gfCNCPoint2[23989] = {X 180.1466, Y 22.4199, Z -3.0000, A 0.000, B 0.000, C 0.000 }
gfCNCPoint2[23990] = {X 179.6136, Y 22.9696, Z -3.0000, A 0.000, B 0.000, C 0.000 }
gfCNCPoint2[23991] = {X 180.2003, Y 22.9879, Z -3.0000, A 0.000, B 0.000, C 0.000 }
gfCNCPoint2[23992] = {X 182.2741, Y 22.7679, Z -3.0000, A 0.000, B 0.000, C 0.000 }
gfCNCPoint2[23993] = {X 184.3552, Y 22.6339, Z -3.0000, A 0.000, B 0.000, C 0.000 }
gfCNCPoint2[23994] = {X 184.7920, Y 22.6180, Z -3.0000, A 0.000, B 0.000, C 0.000 }
gfCNCPoint2[23995] = {X 185.2288, Y 22.6003, Z -3.0000, A 0.000, B 0.000, C 0.000 }
gfCNCPoint2[23996] = {X 185.1444, Y 20.6021, Z -3.0000, A 0.000, B 0.000, C 0.000 }
gfCNCPoint2[23997] = {X 185.1444, Y 20.6021, Z 0.0000, A 0.000, B 0.000, C 0.000 }
gfCNCPoint2[23998] = {X 185.1444, Y 20.6021, Z 11.0000, A 0.000, B 0.000, C 0.000 }
gfCNCPoint2[23999] = {X 186.2306, Y 37.9128, Z 11.0000, A 0.000, B 0.000, C 0.000 }
gfCNCPoint2[24000] = {X 186.2306, Y 37.9128, Z 0.8333, A 0.000, B 0.000, C 0.000 }
gfCNCPoint2[24001] = {X 187.5931, Y 37.8326, Z 0.4676, A 0.000, B 0.000, C 0.000 }
gfCNCPoint2[24002] = {X 189.4216, Y 37.3852, Z -0.0368, A 0.000, B 0.000, C 0.000 }
gfCNCPoint2[24003] = {X 190.1467, Y 37.0730, Z -0.2483, A 0.000, B 0.000, C 0.000 }
gfCNCPoint2[24004] = {X 190.9837, Y 36.7127, Z -0.4925, A 0.000, B 0.000, C 0.000 }
gfCNCPoint2[24005] = {X 191.6928, Y 36.3239, Z -0.7092, A 0.000, B 0.000, C 0.000 }
gfCNCPoint2[24006] = {X 192.4466, Y 35.8119, Z -0.9533, A 0.000, B 0.000, C 0.000 }
gfCNCPoint2[24007] = {X 192.4699, Y 35.2978, Z -1.0913, A 0.000, B 0.000, C 0.000 }
gfCNCPoint2[24008] = {X 192.6316, Y 34.6339, Z -1.2743, A 0.000, B 0.000, C 0.000 }
gfCNCPoint2[24009] = {X 192.8474, Y 34.1666, Z -1.4123, A 0.000, B 0.000, C 0.000 }
gfCNCPoint2[24010] = {X 192.7390, Y 34.1918, Z -1.4421, A 0.000, B 0.000, C 0.000 }
gfCNCPoint2[24011] = {X 191.4103, Y 34.4420, Z -1.8044, A 0.000, B 0.000, C 0.000 }
gfCNCPoint2[24012] = {X 190.5793, Y 34.5489, Z -2.0289, A 0.000, B 0.000, C 0.000 }
gfCNCPoint2[24013] = {X 189.2271, Y 34.6435, Z -2.3921, A 0.000, B 0.000, C 0.000 }
gfCNCPoint2[24014] = {X 186.9625, Y 34.7826, Z -3.0000, A 0.000, B 0.000, C 0.000 }
gfCNCPoint2[24015] = {X 182.5767, Y 35.0519, Z -3.0000, A 0.000, B 0.000, C 0.000 }
gfCNCPoint2[24016] = {X 181.8176, Y 35.1394, Z -3.0000, A 0.000, B 0.000, C 0.000 }
gfCNCPoint2[24017] = {X 181.0723, Y 35.3075, Z -3.0000, A 0.000, B 0.000, C 0.000 }
gfCNCPoint2[24018] = {X 181.0641, Y 35.3819, Z -3.0000, A 0.000, B 0.000, C 0.000 }
gfCNCPoint2[24019] = {X 181.0641, Y 35.4568, Z -3.0000, A 0.000, B 0.000, C 0.000 }
gfCNCPoint2[24020] = {X 181.1571, Y 36.0001, Z -3.0000, A 0.000, B 0.000, C 0.000 }
gfCNCPoint2[24021] = {X 181.4145, Y 36.4875, Z -3.0000, A 0.000, B 0.000, C 0.000 }
gfCNCPoint2[24022] = {X 181.8107, Y 36.8707, Z -3.0000, A 0.000, B 0.000, C 0.000 }
gfCNCPoint2[24023] = {X 182.4285, Y 37.2234, Z -3.0000, A 0.000, B 0.000, C 0.000 }
gfCNCPoint2[24024] = {X 183.0887, Y 37.4882, Z -3.0000, A 0.000, B 0.000, C 0.000 }
gfCNCPoint2[24025] = {X 184.4959, Y 37.8021, Z -3.0000, A 0.000, B 0.000, C 0.000 }
gfCNCPoint2[24026] = {X 185.9331, Y 37.9178, Z -3.0000, A 0.000, B 0.000, C 0.000 }
gfCNCPoint2[24027] = {X 187.3724, Y 37.8332, Z -3.0000, A 0.000, B 0.000, C 0.000 }
gfCNCPoint2[24028] = {X 188.7860, Y 37.5497, Z -3.0000, A 0.000, B 0.000, C 0.000 }
gfCNCPoint2[24029] = {X 190.1467, Y 37.0730, Z -3.0000, A 0.000, B 0.000, C 0.000 }
gfCNCPoint2[24030] = {X 191.3267, Y 36.4971, Z -3.0000, A 0.000, B 0.000, C 0.000 }
gfCNCPoint2[24031] = {X 192.4466, Y 35.8119, Z -3.0000, A 0.000, B 0.000, C 0.000 }
gfCNCPoint2[24032] = {X 192.5671, Y 34.9698, Z -3.0000, A 0.000, B 0.000, C 0.000 }
gfCNCPoint2[24033] = {X 192.8474, Y 34.1666, Z -3.0000, A 0.000, B 0.000, C 0.000 }
gfCNCPoint2[24034] = {X 192.7390, Y 34.1918, Z -3.0000, A 0.000, B 0.000, C 0.000 }
gfCNCPoint2[24035] = {X 190.9896, Y 34.4688, Z -3.0000, A 0.000, B 0.000, C 0.000 }
gfCNCPoint2[24036] = {X 189.2271, Y 34.6435, Z -3.0000, A 0.000, B 0.000, C 0.000 }
gfCNCPoint2[24037] = {X 186.9625, Y 34.7826, Z -3.0000, A 0.000, B 0.000, C 0.000 }
gfCNCPoint2[24038] = {X 190.9563, Y 34.8065, Z -3.0000, A 0.000, B 0.000, C 0.000 }
gfCNCPoint2[24039] = {X 186.9576, Y 34.7027, Z -3.0000, A 0.000, B 0.000, C 0.000 }
gfCNCPoint2[24040] = {X 182.5718, Y 34.9720, Z -3.0000, A 0.000, B 0.000, C 0.000 }
gfCNCPoint2[24041] = {X 181.7801, Y 35.0647, Z -3.0000, A 0.000, B 0.000, C 0.000 }
gfCNCPoint2[24042] = {X 181.0034, Y 35.2440, Z -3.0000, A 0.000, B 0.000, C 0.000 }
gfCNCPoint2[24043] = {X 180.9865, Y 35.3479, Z -3.0000, A 0.000, B 0.000, C 0.000 }
gfCNCPoint2[24044] = {X 180.9840, Y 35.4530, Z -3.0000, A 0.000, B 0.000, C 0.000 }
gfCNCPoint2[24045] = {X 181.0805, Y 36.0232, Z -3.0000, A 0.000, B 0.000, C 0.000 }
gfCNCPoint2[24046] = {X 181.3499, Y 36.5348, Z -3.0000, A 0.000, B 0.000, C 0.000 }
gfCNCPoint2[24047] = {X 181.7656, Y 36.9368, Z -3.0000, A 0.000, B 0.000, C 0.000 }
gfCNCPoint2[24048] = {X 182.3937, Y 37.2955, Z -3.0000, A 0.000, B 0.000, C 0.000 }
gfCNCPoint2[24049] = {X 183.0650, Y 37.5647, Z -3.0000, A 0.000, B 0.000, C 0.000 }
gfCNCPoint2[24050] = {X 184.4832, Y 37.8811, Z -3.0000, A 0.000, B 0.000, C 0.000 }
gfCNCPoint2[24051] = {X 185.9316, Y 37.9978, Z -3.0000, A 0.000, B 0.000, C 0.000 }
gfCNCPoint2[24052] = {X 187.3822, Y 37.9125, Z -3.0000, A 0.000, B 0.000, C 0.000 }
gfCNCPoint2[24053] = {X 188.8070, Y 37.6269, Z -3.0000, A 0.000, B 0.000, C 0.000 }
gfCNCPoint2[24054] = {X 190.1784, Y 37.1465, Z -3.0000, A 0.000, B 0.000, C 0.000 }
gfCNCPoint2[24055] = {X 191.3828, Y 36.5576, Z -3.0000, A 0.000, B 0.000, C 0.000 }
gfCNCPoint2[24056] = {X 192.5249, Y 35.8554, Z -3.0000, A 0.000, B 0.000, C 0.000 }
gfCNCPoint2[24057] = {X 192.6603, Y 34.9271, Z -3.0000, A 0.000, B 0.000, C 0.000 }
gfCNCPoint2[24058] = {X 192.9929, Y 34.0499, Z -3.0000, A 0.000, B 0.000, C 0.000 }
gfCNCPoint2[24059] = {X 192.7315, Y 34.1118, Z -3.0000, A 0.000, B 0.000, C 0.000 }
gfCNCPoint2[24060] = {X 190.9841, Y 34.3888, Z -3.0000, A 0.000, B 0.000, C 0.000 }
gfCNCPoint2[24061] = {X 189.2235, Y 34.5636, Z -3.0000, A 0.000, B 0.000, C 0.000 }
gfCNCPoint2[24062] = {X 186.9576, Y 34.7027, Z -3.0000, A 0.000, B 0.000, C 0.000 }
gfCNCPoint2[24063] = {X 183.0017, Y 35.2949, Z -3.0000, A 0.000, B 0.000, C 0.000 }
gfCNCPoint2[24064] = {X 190.9514, Y 34.7266, Z -3.0000, A 0.000, B 0.000, C 0.000 }
gfCNCPoint2[24065] = {X 186.9527, Y 34.6229, Z -3.0000, A 0.000, B 0.000, C 0.000 }
gfCNCPoint2[24066] = {X 182.5669, Y 34.8922, Z -3.0000, A 0.000, B 0.000, C 0.000 }
gfCNCPoint2[24067] = {X 181.7440, Y 34.9898, Z -3.0000, A 0.000, B 0.000, C 0.000 }
gfCNCPoint2[24068] = {X 180.9376, Y 35.1800, Z -3.0000, A 0.000, B 0.000, C 0.000 }
gfCNCPoint2[24069] = {X 180.9095, Y 35.3162, Z -3.0000, A 0.000, B 0.000, C 0.000 }
gfCNCPoint2[24070] = {X 180.9041, Y 35.4551, Z -3.0000, A 0.000, B 0.000, C 0.000 }
gfCNCPoint2[24071] = {X 181.0051, Y 36.0500, Z -3.0000, A 0.000, B 0.000, C 0.000 }
gfCNCPoint2[24072] = {X 181.2866, Y 36.5836, Z -3.0000, A 0.000, B 0.000, C 0.000 }
gfCNCPoint2[24073] = {X 181.7205, Y 37.0029, Z -3.0000, A 0.000, B 0.000, C 0.000 }
gfCNCPoint2[24074] = {X 182.3589, Y 37.3675, Z -3.0000, A 0.000, B 0.000, C 0.000 }
gfCNCPoint2[24075] = {X 183.0413, Y 37.6411, Z -3.0000, A 0.000, B 0.000, C 0.000 }
gfCNCPoint2[24076] = {X 184.4705, Y 37.9601, Z -3.0000, A 0.000, B 0.000, C 0.000 }
gfCNCPoint2[24077] = {X 185.9302, Y 38.0778, Z -3.0000, A 0.000, B 0.000, C 0.000 }
gfCNCPoint2[24078] = {X 187.3921, Y 37.9919, Z -3.0000, A 0.000, B 0.000, C 0.000 }
gfCNCPoint2[24079] = {X 188.8279, Y 37.7041, Z -3.0000, A 0.000, B 0.000, C 0.000 }
gfCNCPoint2[24080] = {X 190.2100, Y 37.2200, Z -3.0000, A 0.000, B 0.000, C 0.000 }
gfCNCPoint2[24081] = {X 191.4392, Y 36.6179, Z -3.0000, A 0.000, B 0.000, C 0.000 }
gfCNCPoint2[24082] = {X 192.6036, Y 35.8985, Z -3.0000, A 0.000, B 0.000, C 0.000 }
gfCNCPoint2[24083] = {X 192.6773, Y 35.2160, Z -3.0000, A 0.000, B 0.000, C 0.000 }
gfCNCPoint2[24084] = {X 192.8602, Y 34.5544, Z -3.0000, A 0.000, B 0.000, C 0.000 }
gfCNCPoint2[24085] = {X 193.1474, Y 33.9310, Z -3.0000, A 0.000, B 0.000, C 0.000 }
gfCNCPoint2[24086] = {X 192.7149, Y 34.0336, Z -3.0000, A 0.000, B 0.000, C 0.000 }
gfCNCPoint2[24087] = {X 190.9732, Y 34.3096, Z -3.0000, A 0.000, B 0.000, C 0.000 }
gfCNCPoint2[24088] = {X 189.2183, Y 34.4838, Z -3.0000, A 0.000, B 0.000, C 0.000 }
gfCNCPoint2[24089] = {X 186.9527, Y 34.6229, Z -3.0000, A 0.000, B 0.000, C 0.000 }
gfCNCPoint2[24090] = {X 182.9968, Y 35.2151, Z -3.0000, A 0.000, B 0.000, C 0.000 }
gfCNCPoint2[24091] = {X 190.9465, Y 34.6468, Z -3.0000, A 0.000, B 0.000, C 0.000 }
gfCNCPoint2[24092] = {X 186.9478, Y 34.5430, Z -3.0000, A 0.000, B 0.000, C 0.000 }
gfCNCPoint2[24093] = {X 182.5620, Y 34.8123, Z -3.0000, A 0.000, B 0.000, C 0.000 }
gfCNCPoint2[24094] = {X 181.7093, Y 34.9147, Z -3.0000, A 0.000, B 0.000, C 0.000 }
gfCNCPoint2[24095] = {X 180.8742, Y 35.1154, Z -3.0000, A 0.000, B 0.000, C 0.000 }
gfCNCPoint2[24096] = {X 180.8331, Y 35.2840, Z -3.0000, A 0.000, B 0.000, C 0.000 }
gfCNCPoint2[24097] = {X 180.8241, Y 35.4572, Z -3.0000, A 0.000, B 0.000, C 0.000 }
gfCNCPoint2[24098] = {X 180.9297, Y 36.0768, Z -3.0000, A 0.000, B 0.000, C 0.000 }
gfCNCPoint2[24099] = {X 181.2232, Y 36.6325, Z -3.0000, A 0.000, B 0.000, C 0.000 }
gfCNCPoint2[24100] = {X 181.6754, Y 37.0690, Z -3.0000, A 0.000, B 0.000, C 0.000 }
gfCNCPoint2[24101] = {X 182.3241, Y 37.4395, Z -3.0000, A 0.000, B 0.000, C 0.000 }
gfCNCPoint2[24102] = {X 183.0176, Y 37.7175, Z -3.0000, A 0.000, B 0.000, C 0.000 }
gfCNCPoint2[24103] = {X 184.4578, Y 38.0391, Z -3.0000, A 0.000, B 0.000, C 0.000 }
gfCNCPoint2[24104] = {X 185.9288, Y 38.1578, Z -3.0000, A 0.000, B 0.000, C 0.000 }
gfCNCPoint2[24105] = {X 187.4020, Y 38.0713, Z -3.0000, A 0.000, B 0.000, C 0.000 }
gfCNCPoint2[24106] = {X 188.8489, Y 37.7813, Z -3.0000, A 0.000, B 0.000, C 0.000 }
gfCNCPoint2[24107] = {X 190.2416, Y 37.2935, Z -3.0000, A 0.000, B 0.000, C 0.000 }
gfCNCPoint2[24108] = {X 191.4958, Y 36.6780, Z -3.0000, A 0.000, B 0.000, C 0.000 }
gfCNCPoint2[24109] = {X 192.6827, Y 35.9411, Z -3.0000, A 0.000, B 0.000, C 0.000 }
gfCNCPoint2[24110] = {X 192.7627, Y 35.1965, Z -3.0000, A 0.000, B 0.000, C 0.000 }
gfCNCPoint2[24111] = {X 192.9748, Y 34.4783, Z -3.0000, A 0.000, B 0.000, C 0.000 }
gfCNCPoint2[24112] = {X 193.3123, Y 33.8097, Z -3.0000, A 0.000, B 0.000, C 0.000 }
gfCNCPoint2[24113] = {X 192.6983, Y 33.9553, Z -3.0000, A 0.000, B 0.000, C 0.000 }
gfCNCPoint2[24114] = {X 190.9622, Y 34.2303, Z -3.0000, A 0.000, B 0.000, C 0.000 }
gfCNCPoint2[24115] = {X 189.2131, Y 34.4039, Z -3.0000, A 0.000, B 0.000, C 0.000 }
gfCNCPoint2[24116] = {X 186.9478, Y 34.5430, Z -3.0000, A 0.000, B 0.000, C 0.000 }
gfCNCPoint2[24117] = {X 182.9919, Y 35.1352, Z -3.0000, A 0.000, B 0.000, C 0.000 }
gfCNCPoint2[24118] = {X 190.9415, Y 34.5669, Z -3.0000, A 0.000, B 0.000, C 0.000 }
gfCNCPoint2[24119] = {X 186.9429, Y 34.4632, Z -3.0000, A 0.000, B 0.000, C 0.000 }
gfCNCPoint2[24120] = {X 182.5571, Y 34.7325, Z -3.0000, A 0.000, B 0.000, C 0.000 }
gfCNCPoint2[24121] = {X 181.6755, Y 34.8395, Z -3.0000, A 0.000, B 0.000, C 0.000 }
gfCNCPoint2[24122] = {X 180.8129, Y 35.0505, Z -3.0000, A 0.000, B 0.000, C 0.000 }
gfCNCPoint2[24123] = {X 180.7572, Y 35.2513, Z -3.0000, A 0.000, B 0.000, C 0.000 }
gfCNCPoint2[24124] = {X 180.7441, Y 35.4593, Z -3.0000, A 0.000, B 0.000, C 0.000 }
gfCNCPoint2[24125] = {X 180.8543, Y 36.1035, Z -3.0000, A 0.000, B 0.000, C 0.000 }
gfCNCPoint2[24126] = {X 181.1598, Y 36.6813, Z -3.0000, A 0.000, B 0.000, C 0.000 }
gfCNCPoint2[24127] = {X 181.6303, Y 37.1351, Z -3.0000, A 0.000, B 0.000, C 0.000 }
gfCNCPoint2[24128] = {X 182.2893, Y 37.5116, Z -3.0000, A 0.000, B 0.000, C 0.000 }
gfCNCPoint2[24129] = {X 182.9939, Y 37.7939, Z -3.0000, A 0.000, B 0.000, C 0.000 }
gfCNCPoint2[24130] = {X 184.4452, Y 38.1181, Z -3.0000, A 0.000, B 0.000, C 0.000 }
gfCNCPoint2[24131] = {X 185.9274, Y 38.2378, Z -3.0000, A 0.000, B 0.000, C 0.000 }
gfCNCPoint2[24132] = {X 187.4118, Y 38.1507, Z -3.0000, A 0.000, B 0.000, C 0.000 }
gfCNCPoint2[24133] = {X 188.8699, Y 37.8585, Z -3.0000, A 0.000, B 0.000, C 0.000 }
gfCNCPoint2[24134] = {X 190.2733, Y 37.3669, Z -3.0000, A 0.000, B 0.000, C 0.000 }
gfCNCPoint2[24135] = {X 191.5527, Y 36.7379, Z -3.0000, A 0.000, B 0.000, C 0.000 }
gfCNCPoint2[24136] = {X 192.7622, Y 35.9833, Z -3.0000, A 0.000, B 0.000, C 0.000 }
gfCNCPoint2[24137] = {X 192.8359, Y 35.2389, Z -3.0000, A 0.000, B 0.000, C 0.000 }
gfCNCPoint2[24138] = {X 193.0442, Y 34.5204, Z -3.0000, A 0.000, B 0.000, C 0.000 }
gfCNCPoint2[24139] = {X 193.3801, Y 33.8520, Z -3.0000, A 0.000, B 0.000, C 0.000 }
gfCNCPoint2[24140] = {X 193.4231, Y 33.7847, Z -3.0000, A 0.000, B 0.000, C 0.000 }
gfCNCPoint2[24141] = {X 193.4673, Y 33.7182, Z -3.0000, A 0.000, B 0.000, C 0.000 }
gfCNCPoint2[24142] = {X 193.3655, Y 33.7149, Z -3.0000, A 0.000, B 0.000, C 0.000 }
gfCNCPoint2[24143] = {X 192.6816, Y 33.8770, Z -3.0000, A 0.000, B 0.000, C 0.000 }
gfCNCPoint2[24144] = {X 190.9512, Y 34.1511, Z -3.0000, A 0.000, B 0.000, C 0.000 }
gfCNCPoint2[24145] = {X 189.2078, Y 34.3241, Z -3.0000, A 0.000, B 0.000, C 0.000 }
gfCNCPoint2[24146] = {X 186.9429, Y 34.4632, Z -3.0000, A 0.000, B 0.000, C 0.000 }
gfCNCPoint2[24147] = {X 182.9870, Y 35.0554, Z -3.0000, A 0.000, B 0.000, C 0.000 }
gfCNCPoint2[24148] = {X 190.9366, Y 34.4871, Z -3.0000, A 0.000, B 0.000, C 0.000 }
gfCNCPoint2[24149] = {X 186.9380, Y 34.3833, Z -3.0000, A 0.000, B 0.000, C 0.000 }
gfCNCPoint2[24150] = {X 182.5522, Y 34.6526, Z -3.0000, A 0.000, B 0.000, C 0.000 }
gfCNCPoint2[24151] = {X 181.6426, Y 34.7642, Z -3.0000, A 0.000, B 0.000, C 0.000 }
gfCNCPoint2[24152] = {X 180.7533, Y 34.9853, Z -3.0000, A 0.000, B 0.000, C 0.000 }
gfCNCPoint2[24153] = {X 180.6819, Y 35.2183, Z -3.0000, A 0.000, B 0.000, C 0.000 }
gfCNCPoint2[24154] = {X 180.6641, Y 35.4613, Z -3.0000, A 0.000, B 0.000, C 0.000 }
gfCNCPoint2[24155] = {X 180.7789, Y 36.1303, Z -3.0000, A 0.000, B 0.000, C 0.000 }
gfCNCPoint2[24156] = {X 181.0965, Y 36.7302, Z -3.0000, A 0.000, B 0.000, C 0.000 }
gfCNCPoint2[24157] = {X 181.5852, Y 37.2012, Z -3.0000, A 0.000, B 0.000, C 0.000 }
gfCNCPoint2[24158] = {X 182.2546, Y 37.5836, Z -3.0000, A 0.000, B 0.000, C 0.000 }
gfCNCPoint2[24159] = {X 182.9702, Y 37.8703, Z -3.0000, A 0.000, B 0.000, C 0.000 }
gfCNCPoint2[24160] = {X 184.4325, Y 38.1971, Z -3.0000, A 0.000, B 0.000, C 0.000 }
gfCNCPoint2[24161] = {X 185.9259, Y 38.3178, Z -3.0000, A 0.000, B 0.000, C 0.000 }
gfCNCPoint2[24162] = {X 187.4217, Y 38.2301, Z -3.0000, A 0.000, B 0.000, C 0.000 }
gfCNCPoint2[24163] = {X 188.8908, Y 37.9358, Z -3.0000, A 0.000, B 0.000, C 0.000 }
gfCNCPoint2[24164] = {X 190.3049, Y 37.4404, Z -3.0000, A 0.000, B 0.000, C 0.000 }
gfCNCPoint2[24165] = {X 191.6098, Y 36.7977, Z -3.0000, A 0.000, B 0.000, C 0.000 }
gfCNCPoint2[24166] = {X 192.8422, Y 36.0250, Z -3.0000, A 0.000, B 0.000, C 0.000 }
gfCNCPoint2[24167] = {X 192.9290, Y 35.1818, Z -3.0000, A 0.000, B 0.000, C 0.000 }
gfCNCPoint2[24168] = {X 193.1917, Y 34.3757, Z -3.0000, A 0.000, B 0.000, C 0.000 }
gfCNCPoint2[24169] = {X 193.6183, Y 33.6431, Z -3.0000, A 0.000, B 0.000, C 0.000 }
gfCNCPoint2[24170] = {X 193.3575, Y 33.6346, Z -3.0000, A 0.000, B 0.000, C 0.000 }
gfCNCPoint2[24171] = {X 192.6650, Y 33.7987, Z -3.0000, A 0.000, B 0.000, C 0.000 }
gfCNCPoint2[24172] = {X 190.9402, Y 34.0718, Z -3.0000, A 0.000, B 0.000, C 0.000 }
gfCNCPoint2[24173] = {X 189.2026, Y 34.2443, Z -3.0000, A 0.000, B 0.000, C 0.000 }
gfCNCPoint2[24174] = {X 186.9380, Y 34.3833, Z -3.0000, A 0.000, B 0.000, C 0.000 }
gfCNCPoint2[24175] = {X 182.9821, Y 34.9755, Z -3.0000, A 0.000, B 0.000, C 0.000 }
gfCNCPoint2[24176] = {X 182.9821, Y 34.9755, Z 0.0000, A 0.000, B 0.000, C 0.000 }
gfCNCPoint2[24177] = {X 182.9821, Y 34.9755, Z 11.0000, A 0.000, B 0.000, C 0.000 }
gfCNCPoint2[24178] = {X 165.6772, Y 73.8165, Z 11.0000, A 0.000, B 0.000, C 0.000 }
gfCNCPoint2[24179] = {X 165.6772, Y 73.8165, Z 0.8333, A 0.000, B 0.000, C 0.000 }
gfCNCPoint2[24180] = {X 161.3996, Y 78.5670, Z -0.8796, A 0.000, B 0.000, C 0.000 }
gfCNCPoint2[24181] = {X 169.3132, Y 78.5670, Z -3.0000, A 0.000, B 0.000, C 0.000 }
gfCNCPoint2[24182] = {X 169.3132, Y 76.1670, Z -3.0000, A 0.000, B 0.000, C 0.000 }
gfCNCPoint2[24183] = {X 171.8361, Y 76.1670, Z -3.0000, A 0.000, B 0.000, C 0.000 }
gfCNCPoint2[24184] = {X 169.3147, Y 73.3634, Z -3.0000, A 0.000, B 0.000, C 0.000 }
gfCNCPoint2[24185] = {X 166.7903, Y 76.1670, Z -3.0000, A 0.000, B 0.000, C 0.000 }
gfCNCPoint2[24186] = {X 169.3132, Y 76.1670, Z -3.0000, A 0.000, B 0.000, C 0.000 }
gfCNCPoint2[24187] = {X 169.3132, Y 78.5670, Z -3.0000, A 0.000, B 0.000, C 0.000 }
gfCNCPoint2[24188] = {X 177.2224, Y 78.5670, Z -3.0000, A 0.000, B 0.000, C 0.000 }
gfCNCPoint2[24189] = {X 169.3158, Y 69.7756, Z -3.0000, A 0.000, B 0.000, C 0.000 }
gfCNCPoint2[24190] = {X 161.3996, Y 78.5670, Z -3.0000, A 0.000, B 0.000, C 0.000 }
gfCNCPoint2[24191] = {X 169.3132, Y 78.5670, Z -3.0000, A 0.000, B 0.000, C 0.000 }
gfCNCPoint2[24192] = {X 169.3132, Y 74.6470, Z -3.0000, A 0.000, B 0.000, C 0.000 }
gfCNCPoint2[24193] = {X 169.3132, Y 78.6470, Z -3.0000, A 0.000, B 0.000, C 0.000 }
gfCNCPoint2[24194] = {X 177.4019, Y 78.6470, Z -3.0000, A 0.000, B 0.000, C 0.000 }
gfCNCPoint2[24195] = {X 169.3159, Y 69.6560, Z -3.0000, A 0.000, B 0.000, C 0.000 }
gfCNCPoint2[24196] = {X 161.2199, Y 78.6470, Z -3.0000, A 0.000, B 0.000, C 0.000 }
gfCNCPoint2[24197] = {X 169.3132, Y 78.6470, Z -3.0000, A 0.000, B 0.000, C 0.000 }
gfCNCPoint2[24198] = {X 169.3132, Y 74.6470, Z -3.0000, A 0.000, B 0.000, C 0.000 }
gfCNCPoint2[24199] = {X 169.3132, Y 74.7270, Z -3.0000, A 0.000, B 0.000, C 0.000 }
gfCNCPoint2[24200] = {X 169.3132, Y 78.7270, Z -3.0000, A 0.000, B 0.000, C 0.000 }
gfCNCPoint2[24201] = {X 177.5814, Y 78.7270, Z -3.0000, A 0.000, B 0.000, C 0.000 }
gfCNCPoint2[24202] = {X 169.3159, Y 69.5364, Z -3.0000, A 0.000, B 0.000, C 0.000 }
gfCNCPoint2[24203] = {X 161.0403, Y 78.7270, Z -3.0000, A 0.000, B 0.000, C 0.000 }
gfCNCPoint2[24204] = {X 169.3132, Y 78.7270, Z -3.0000, A 0.000, B 0.000, C 0.000 }
gfCNCPoint2[24205] = {X 169.3132, Y 74.7270, Z -3.0000, A 0.000, B 0.000, C 0.000 }
gfCNCPoint2[24206] = {X 169.3132, Y 74.8070, Z -3.0000, A 0.000, B 0.000, C 0.000 }
gfCNCPoint2[24207] = {X 169.3132, Y 78.8070, Z -3.0000, A 0.000, B 0.000, C 0.000 }
gfCNCPoint2[24208] = {X 177.7610, Y 78.8070, Z -3.0000, A 0.000, B 0.000, C 0.000 }
gfCNCPoint2[24209] = {X 169.3159, Y 69.4168, Z -3.0000, A 0.000, B 0.000, C 0.000 }
gfCNCPoint2[24210] = {X 160.8606, Y 78.8070, Z -3.0000, A 0.000, B 0.000, C 0.000 }
gfCNCPoint2[24211] = {X 169.3132, Y 78.8070, Z -3.0000, A 0.000, B 0.000, C 0.000 }
gfCNCPoint2[24212] = {X 169.3132, Y 74.8070, Z -3.0000, A 0.000, B 0.000, C 0.000 }
gfCNCPoint2[24213] = {X 169.3132, Y 74.8870, Z -3.0000, A 0.000, B 0.000, C 0.000 }
gfCNCPoint2[24214] = {X 169.3132, Y 78.8870, Z -3.0000, A 0.000, B 0.000, C 0.000 }
gfCNCPoint2[24215] = {X 177.9405, Y 78.8870, Z -3.0000, A 0.000, B 0.000, C 0.000 }
gfCNCPoint2[24216] = {X 169.3160, Y 69.2972, Z -3.0000, A 0.000, B 0.000, C 0.000 }
gfCNCPoint2[24217] = {X 160.6809, Y 78.8870, Z -3.0000, A 0.000, B 0.000, C 0.000 }
gfCNCPoint2[24218] = {X 169.3132, Y 78.8870, Z -3.0000, A 0.000, B 0.000, C 0.000 }
gfCNCPoint2[24219] = {X 169.3132, Y 74.8870, Z -3.0000, A 0.000, B 0.000, C 0.000 }
gfCNCPoint2[24220] = {X 169.3132, Y 74.9670, Z -3.0000, A 0.000, B 0.000, C 0.000 }
gfCNCPoint2[24221] = {X 169.3132, Y 78.9670, Z -3.0000, A 0.000, B 0.000, C 0.000 }
gfCNCPoint2[24222] = {X 178.1201, Y 78.9670, Z -3.0000, A 0.000, B 0.000, C 0.000 }
gfCNCPoint2[24223] = {X 169.3160, Y 69.1776, Z -3.0000, A 0.000, B 0.000, C 0.000 }
gfCNCPoint2[24224] = {X 160.5012, Y 78.9670, Z -3.0000, A 0.000, B 0.000, C 0.000 }
gfCNCPoint2[24225] = {X 169.3132, Y 78.9670, Z -3.0000, A 0.000, B 0.000, C 0.000 }
gfCNCPoint2[24226] = {X 169.3132, Y 74.9670, Z -3.0000, A 0.000, B 0.000, C 0.000 }
gfCNCPoint2[24227] = {X 169.3132, Y 74.9670, Z 0.0000, A 0.000, B 0.000, C 0.000 }
gfCNCPoint2[24228] = {X 169.3132, Y 74.9670, Z 11.0000, A 0.000, B 0.000, C 0.000 }
gfCNCPoint2[24229] = {X 11.7108, Y 37.8795, Z 11.0000, A 0.000, B 0.000, C 0.000 }
gfCNCPoint2[24230] = {X 11.7108, Y 37.8795, Z 0.8333, A 0.000, B 0.000, C 0.000 }
gfCNCPoint2[24231] = {X 12.4946, Y 37.9514, Z 0.6224, A 0.000, B 0.000, C 0.000 }
gfCNCPoint2[24232] = {X 14.1356, Y 37.8409, Z 0.1817, A 0.000, B 0.000, C 0.000 }
gfCNCPoint2[24233] = {X 15.7386, Y 37.4728, Z -0.2590, A 0.000, B 0.000, C 0.000 }
gfCNCPoint2[24234] = {X 16.4708, Y 37.1794, Z -0.4703, A 0.000, B 0.000, C 0.000 }
gfCNCPoint2[24235] = {X 17.3029, Y 36.8460, Z -0.7105, A 0.000, B 0.000, C 0.000 }
gfCNCPoint2[24236] = {X 18.2940, Y 36.3175, Z -1.0115, A 0.000, B 0.000, C 0.000 }
gfCNCPoint2[24237] = {X 19.0345, Y 35.8124, Z -1.2517, A 0.000, B 0.000, C 0.000 }
gfCNCPoint2[24238] = {X 19.0577, Y 35.2982, Z -1.3896, A 0.000, B 0.000, C 0.000 }
gfCNCPoint2[24239] = {X 19.2191, Y 34.6349, Z -1.5725, A 0.000, B 0.000, C 0.000 }
gfCNCPoint2[24240] = {X 19.4347, Y 34.1676, Z -1.7104, A 0.000, B 0.000, C 0.000 }
gfCNCPoint2[24241] = {X 18.1976, Y 34.4161, Z -2.0485, A 0.000, B 0.000, C 0.000 }
gfCNCPoint2[24242] = {X 17.3693, Y 34.5286, Z -2.2725, A 0.000, B 0.000, C 0.000 }
gfCNCPoint2[24243] = {X 16.1107, Y 34.6189, Z -2.6106, A 0.000, B 0.000, C 0.000 }
gfCNCPoint2[24244] = {X 15.3860, Y 34.6726, Z -2.8053, A 0.000, B 0.000, C 0.000 }
gfCNCPoint2[24245] = {X 14.6610, Y 34.7222, Z -3.0000, A 0.000, B 0.000, C 0.000 }
gfCNCPoint2[24246] = {X 12.2608, Y 34.8748, Z -3.0000, A 0.000, B 0.000, C 0.000 }
gfCNCPoint2[24247] = {X 9.8593, Y 35.0045, Z -3.0000, A 0.000, B 0.000, C 0.000 }
gfCNCPoint2[24248] = {X 8.7533, Y 35.0948, Z -3.0000, A 0.000, B 0.000, C 0.000 }
gfCNCPoint2[24249] = {X 7.6646, Y 35.3089, Z -3.0000, A 0.000, B 0.000, C 0.000 }
gfCNCPoint2[24250] = {X 7.6549, Y 35.3709, Z -3.0000, A 0.000, B 0.000, C 0.000 }
gfCNCPoint2[24251] = {X 7.6516, Y 35.4334, Z -3.0000, A 0.000, B 0.000, C 0.000 }
gfCNCPoint2[24252] = {X 7.7522, Y 36.0266, Z -3.0000, A 0.000, B 0.000, C 0.000 }
gfCNCPoint2[24253] = {X 8.0469, Y 36.5510, Z -3.0000, A 0.000, B 0.000, C 0.000 }
gfCNCPoint2[24254] = {X 8.5011, Y 36.9455, Z -3.0000, A 0.000, B 0.000, C 0.000 }
gfCNCPoint2[24255] = {X 9.2719, Y 37.3362, Z -3.0000, A 0.000, B 0.000, C 0.000 }
gfCNCPoint2[24256] = {X 10.0919, Y 37.6087, Z -3.0000, A 0.000, B 0.000, C 0.000 }
gfCNCPoint2[24257] = {X 11.3690, Y 37.8462, Z -3.0000, A 0.000, B 0.000, C 0.000 }
gfCNCPoint2[24258] = {X 12.6659, Y 37.9220, Z -3.0000, A 0.000, B 0.000, C 0.000 }
gfCNCPoint2[24259] = {X 13.9620, Y 37.8348, Z -3.0000, A 0.000, B 0.000, C 0.000 }
gfCNCPoint2[24260] = {X 15.2370, Y 37.5859, Z -3.0000, A 0.000, B 0.000, C 0.000 }
gfCNCPoint2[24261] = {X 16.4708, Y 37.1794, Z -3.0000, A 0.000, B 0.000, C 0.000 }
gfCNCPoint2[24262] = {X 17.7899, Y 36.5657, Z -3.0000, A 0.000, B 0.000, C 0.000 }
gfCNCPoint2[24263] = {X 19.0345, Y 35.8124, Z -3.0000, A 0.000, B 0.000, C 0.000 }
gfCNCPoint2[24264] = {X 19.1548, Y 34.9706, Z -3.0000, A 0.000, B 0.000, C 0.000 }
gfCNCPoint2[24265] = {X 19.4347, Y 34.1676, Z -3.0000, A 0.000, B 0.000, C 0.000 }
gfCNCPoint2[24266] = {X 17.7799, Y 34.4459, Z -3.0000, A 0.000, B 0.000, C 0.000 }
gfCNCPoint2[24267] = {X 16.1107, Y 34.6189, Z -3.0000, A 0.000, B 0.000, C 0.000 }
gfCNCPoint2[24268] = {X 15.3859, Y 34.6716, Z -3.0000, A 0.000, B 0.000, C 0.000 }
gfCNCPoint2[24269] = {X 14.6610, Y 34.7222, Z -3.0000, A 0.000, B 0.000, C 0.000 }
gfCNCPoint2[24270] = {X 18.6548, Y 34.7184, Z -3.0000, A 0.000, B 0.000, C 0.000 }
gfCNCPoint2[24271] = {X 14.6556, Y 34.6424, Z -3.0000, A 0.000, B 0.000, C 0.000 }
gfCNCPoint2[24272] = {X 12.2590, Y 34.7948, Z -3.0000, A 0.000, B 0.000, C 0.000 }
gfCNCPoint2[24273] = {X 9.8611, Y 34.9245, Z -3.0000, A 0.000, B 0.000, C 0.000 }
gfCNCPoint2[24274] = {X 8.7205, Y 35.0186, Z -3.0000, A 0.000, B 0.000, C 0.000 }
gfCNCPoint2[24275] = {X 7.5984, Y 35.2434, Z -3.0000, A 0.000, B 0.000, C 0.000 }
gfCNCPoint2[24276] = {X 7.5785, Y 35.3374, Z -3.0000, A 0.000, B 0.000, C 0.000 }
gfCNCPoint2[24277] = {X 7.5716, Y 35.4331, Z -3.0000, A 0.000, B 0.000, C 0.000 }
gfCNCPoint2[24278] = {X 7.6768, Y 36.0532, Z -3.0000, A 0.000, B 0.000, C 0.000 }
gfCNCPoint2[24279] = {X 7.9849, Y 36.6016, Z -3.0000, A 0.000, B 0.000, C 0.000 }
gfCNCPoint2[24280] = {X 8.4598, Y 37.0140, Z -3.0000, A 0.000, B 0.000, C 0.000 }
gfCNCPoint2[24281] = {X 9.2411, Y 37.4100, Z -3.0000, A 0.000, B 0.000, C 0.000 }
gfCNCPoint2[24282] = {X 10.0723, Y 37.6863, Z -3.0000, A 0.000, B 0.000, C 0.000 }
gfCNCPoint2[24283] = {X 11.3593, Y 37.9257, Z -3.0000, A 0.000, B 0.000, C 0.000 }
gfCNCPoint2[24284] = {X 12.6662, Y 38.0020, Z -3.0000, A 0.000, B 0.000, C 0.000 }
gfCNCPoint2[24285] = {X 13.9724, Y 37.9141, Z -3.0000, A 0.000, B 0.000, C 0.000 }
gfCNCPoint2[24286] = {X 15.2572, Y 37.6633, Z -3.0000, A 0.000, B 0.000, C 0.000 }
gfCNCPoint2[24287] = {X 16.5006, Y 37.2537, Z -3.0000, A 0.000, B 0.000, C 0.000 }
gfCNCPoint2[24288] = {X 17.8453, Y 36.6268, Z -3.0000, A 0.000, B 0.000, C 0.000 }
gfCNCPoint2[24289] = {X 19.1128, Y 35.8557, Z -3.0000, A 0.000, B 0.000, C 0.000 }
gfCNCPoint2[24290] = {X 19.2471, Y 34.9310, Z -3.0000, A 0.000, B 0.000, C 0.000 }
gfCNCPoint2[24291] = {X 19.5772, Y 34.0569, Z -3.0000, A 0.000, B 0.000, C 0.000 }
gfCNCPoint2[24292] = {X 17.8490, Y 34.3556, Z -3.0000, A 0.000, B 0.000, C 0.000 }
gfCNCPoint2[24293] = {X 16.1049, Y 34.5391, Z -3.0000, A 0.000, B 0.000, C 0.000 }
gfCNCPoint2[24294] = {X 15.3803, Y 34.5918, Z -3.0000, A 0.000, B 0.000, C 0.000 }
gfCNCPoint2[24295] = {X 14.6556, Y 34.6424, Z -3.0000, A 0.000, B 0.000, C 0.000 }
gfCNCPoint2[24296] = {X 10.7039, Y 35.2621, Z -3.0000, A 0.000, B 0.000, C 0.000 }
gfCNCPoint2[24297] = {X 18.6494, Y 34.6385, Z -3.0000, A 0.000, B 0.000, C 0.000 }
gfCNCPoint2[24298] = {X 14.6501, Y 34.5626, Z -3.0000, A 0.000, B 0.000, C 0.000 }
gfCNCPoint2[24299] = {X 12.2548, Y 34.7149, Z -3.0000, A 0.000, B 0.000, C 0.000 }
gfCNCPoint2[24300] = {X 9.8581, Y 34.8445, Z -3.0000, A 0.000, B 0.000, C 0.000 }
gfCNCPoint2[24301] = {X 8.6870, Y 34.9426, Z -3.0000, A 0.000, B 0.000, C 0.000 }
gfCNCPoint2[24302] = {X 7.5354, Y 35.1773, Z -3.0000, A 0.000, B 0.000, C 0.000 }
gfCNCPoint2[24303] = {X 7.5028, Y 35.3032, Z -3.0000, A 0.000, B 0.000, C 0.000 }
gfCNCPoint2[24304] = {X 7.4916, Y 35.4328, Z -3.0000, A 0.000, B 0.000, C 0.000 }
gfCNCPoint2[24305] = {X 7.6014, Y 36.0799, Z -3.0000, A 0.000, B 0.000, C 0.000 }
gfCNCPoint2[24306] = {X 7.9229, Y 36.6521, Z -3.0000, A 0.000, B 0.000, C 0.000 }
gfCNCPoint2[24307] = {X 8.4184, Y 37.0825, Z -3.0000, A 0.000, B 0.000, C 0.000 }
gfCNCPoint2[24308] = {X 9.2103, Y 37.4839, Z -3.0000, A 0.000, B 0.000, C 0.000 }
gfCNCPoint2[24309] = {X 10.0528, Y 37.7638, Z -3.0000, A 0.000, B 0.000, C 0.000 }
gfCNCPoint2[24310] = {X 11.3497, Y 38.0051, Z -3.0000, A 0.000, B 0.000, C 0.000 }
gfCNCPoint2[24311] = {X 12.6666, Y 38.0820, Z -3.0000, A 0.000, B 0.000, C 0.000 }
gfCNCPoint2[24312] = {X 13.9827, Y 37.9934, Z -3.0000, A 0.000, B 0.000, C 0.000 }
gfCNCPoint2[24313] = {X 15.2774, Y 37.7408, Z -3.0000, A 0.000, B 0.000, C 0.000 }
gfCNCPoint2[24314] = {X 16.5303, Y 37.3279, Z -3.0000, A 0.000, B 0.000, C 0.000 }
gfCNCPoint2[24315] = {X 17.9009, Y 36.6877, Z -3.0000, A 0.000, B 0.000, C 0.000 }
gfCNCPoint2[24316] = {X 19.1915, Y 35.8986, Z -3.0000, A 0.000, B 0.000, C 0.000 }
gfCNCPoint2[24317] = {X 19.2643, Y 35.2208, Z -3.0000, A 0.000, B 0.000, C 0.000 }
gfCNCPoint2[24318] = {X 19.4448, Y 34.5633, Z -3.0000, A 0.000, B 0.000, C 0.000 }
gfCNCPoint2[24319] = {X 19.7283, Y 33.9433, Z -3.0000, A 0.000, B 0.000, C 0.000 }
gfCNCPoint2[24320] = {X 17.9227, Y 34.2645, Z -3.0000, A 0.000, B 0.000, C 0.000 }
gfCNCPoint2[24321] = {X 16.0990, Y 34.4593, Z -3.0000, A 0.000, B 0.000, C 0.000 }
gfCNCPoint2[24322] = {X 15.3747, Y 34.5120, Z -3.0000, A 0.000, B 0.000, C 0.000 }
gfCNCPoint2[24323] = {X 14.6501, Y 34.5626, Z -3.0000, A 0.000, B 0.000, C 0.000 }
gfCNCPoint2[24324] = {X 10.6984, Y 35.1823, Z -3.0000, A 0.000, B 0.000, C 0.000 }
gfCNCPoint2[24325] = {X 18.6439, Y 34.5587, Z -3.0000, A 0.000, B 0.000, C 0.000 }
gfCNCPoint2[24326] = {X 14.6446, Y 34.4828, Z -3.0000, A 0.000, B 0.000, C 0.000 }
gfCNCPoint2[24327] = {X 12.2506, Y 34.6351, Z -3.0000, A 0.000, B 0.000, C 0.000 }
gfCNCPoint2[24328] = {X 9.8552, Y 34.7645, Z -3.0000, A 0.000, B 0.000, C 0.000 }
gfCNCPoint2[24329] = {X 8.6548, Y 34.8664, Z -3.0000, A 0.000, B 0.000, C 0.000 }
gfCNCPoint2[24330] = {X 7.4751, Y 35.1106, Z -3.0000, A 0.000, B 0.000, C 0.000 }
gfCNCPoint2[24331] = {X 7.4279, Y 35.2685, Z -3.0000, A 0.000, B 0.000, C 0.000 }
gfCNCPoint2[24332] = {X 7.4116, Y 35.4326, Z -3.0000, A 0.000, B 0.000, C 0.000 }
gfCNCPoint2[24333] = {X 7.5260, Y 36.1066, Z -3.0000, A 0.000, B 0.000, C 0.000 }
gfCNCPoint2[24334] = {X 7.8609, Y 36.7026, Z -3.0000, A 0.000, B 0.000, C 0.000 }
gfCNCPoint2[24335] = {X 8.3770, Y 37.1510, Z -3.0000, A 0.000, B 0.000, C 0.000 }
gfCNCPoint2[24336] = {X 9.1795, Y 37.5577, Z -3.0000, A 0.000, B 0.000, C 0.000 }
gfCNCPoint2[24337] = {X 10.0333, Y 37.8414, Z -3.0000, A 0.000, B 0.000, C 0.000 }
gfCNCPoint2[24338] = {X 11.3400, Y 38.0845, Z -3.0000, A 0.000, B 0.000, C 0.000 }
gfCNCPoint2[24339] = {X 12.6669, Y 38.1620, Z -3.0000, A 0.000, B 0.000, C 0.000 }
gfCNCPoint2[24340] = {X 13.9931, Y 38.0728, Z -3.0000, A 0.000, B 0.000, C 0.000 }
gfCNCPoint2[24341] = {X 15.2977, Y 37.8182, Z -3.0000, A 0.000, B 0.000, C 0.000 }
gfCNCPoint2[24342] = {X 16.5601, Y 37.4022, Z -3.0000, A 0.000, B 0.000, C 0.000 }
gfCNCPoint2[24343] = {X 17.9567, Y 36.7485, Z -3.0000, A 0.000, B 0.000, C 0.000 }
gfCNCPoint2[24344] = {X 19.2706, Y 35.9411, Z -3.0000, A 0.000, B 0.000, C 0.000 }
gfCNCPoint2[24345] = {X 19.3492, Y 35.2029, Z -3.0000, A 0.000, B 0.000, C 0.000 }
gfCNCPoint2[24346] = {X 19.5579, Y 34.4904, Z -3.0000, A 0.000, B 0.000, C 0.000 }
gfCNCPoint2[24347] = {X 19.8898, Y 33.8263, Z -3.0000, A 0.000, B 0.000, C 0.000 }
gfCNCPoint2[24348] = {X 18.0016, Y 34.1723, Z -3.0000, A 0.000, B 0.000, C 0.000 }
gfCNCPoint2[24349] = {X 16.0932, Y 34.3795, Z -3.0000, A 0.000, B 0.000, C 0.000 }
gfCNCPoint2[24350] = {X 15.3690, Y 34.4322, Z -3.0000, A 0.000, B 0.000, C 0.000 }
gfCNCPoint2[24351] = {X 14.6446, Y 34.4828, Z -3.0000, A 0.000, B 0.000, C 0.000 }
gfCNCPoint2[24352] = {X 10.6929, Y 35.1025, Z -3.0000, A 0.000, B 0.000, C 0.000 }
gfCNCPoint2[24353] = {X 18.6385, Y 34.4789, Z -3.0000, A 0.000, B 0.000, C 0.000 }
gfCNCPoint2[24354] = {X 14.6392, Y 34.4030, Z -3.0000, A 0.000, B 0.000, C 0.000 }
gfCNCPoint2[24355] = {X 12.2464, Y 34.5552, Z -3.0000, A 0.000, B 0.000, C 0.000 }
gfCNCPoint2[24356] = {X 9.8522, Y 34.6846, Z -3.0000, A 0.000, B 0.000, C 0.000 }
gfCNCPoint2[24357] = {X 8.6236, Y 34.7901, Z -3.0000, A 0.000, B 0.000, C 0.000 }
gfCNCPoint2[24358] = {X 7.4169, Y 35.0435, Z -3.0000, A 0.000, B 0.000, C 0.000 }
gfCNCPoint2[24359] = {X 7.3535, Y 35.2333, Z -3.0000, A 0.000, B 0.000, C 0.000 }
gfCNCPoint2[24360] = {X 7.3316, Y 35.4323, Z -3.0000, A 0.000, B 0.000, C 0.000 }
gfCNCPoint2[24361] = {X 7.3983, Y 35.9625, Z -3.0000, A 0.000, B 0.000, C 0.000 }
gfCNCPoint2[24362] = {X 7.5980, Y 36.4582, Z -3.0000, A 0.000, B 0.000, C 0.000 }
gfCNCPoint2[24363] = {X 7.9175, Y 36.8866, Z -3.0000, A 0.000, B 0.000, C 0.000 }
gfCNCPoint2[24364] = {X 8.3357, Y 37.2194, Z -3.0000, A 0.000, B 0.000, C 0.000 }
gfCNCPoint2[24365] = {X 9.1487, Y 37.6315, Z -3.0000, A 0.000, B 0.000, C 0.000 }
gfCNCPoint2[24366] = {X 10.0137, Y 37.9190, Z -3.0000, A 0.000, B 0.000, C 0.000 }
gfCNCPoint2[24367] = {X 11.3303, Y 38.1639, Z -3.0000, A 0.000, B 0.000, C 0.000 }
gfCNCPoint2[24368] = {X 12.6673, Y 38.2420, Z -3.0000, A 0.000, B 0.000, C 0.000 }
gfCNCPoint2[24369] = {X 14.0035, Y 38.1521, Z -3.0000, A 0.000, B 0.000, C 0.000 }
gfCNCPoint2[24370] = {X 15.3179, Y 37.8956, Z -3.0000, A 0.000, B 0.000, C 0.000 }
gfCNCPoint2[24371] = {X 16.5898, Y 37.4764, Z -3.0000, A 0.000, B 0.000, C 0.000 }
gfCNCPoint2[24372] = {X 18.0129, Y 36.8091, Z -3.0000, A 0.000, B 0.000, C 0.000 }
gfCNCPoint2[24373] = {X 19.3501, Y 35.9832, Z -3.0000, A 0.000, B 0.000, C 0.000 }
gfCNCPoint2[24374] = {X 19.4352, Y 35.1814, Z -3.0000, A 0.000, B 0.000, C 0.000 }
gfCNCPoint2[24375] = {X 19.6764, Y 34.4120, Z -3.0000, A 0.000, B 0.000, C 0.000 }
gfCNCPoint2[24376] = {X 20.0641, Y 33.7050, Z -3.0000, A 0.000, B 0.000, C 0.000 }
gfCNCPoint2[24377] = {X 18.0872, Y 34.0788, Z -3.0000, A 0.000, B 0.000, C 0.000 }
gfCNCPoint2[24378] = {X 16.0874, Y 34.2997, Z -3.0000, A 0.000, B 0.000, C 0.000 }
gfCNCPoint2[24379] = {X 15.3634, Y 34.3524, Z -3.0000, A 0.000, B 0.000, C 0.000 }
gfCNCPoint2[24380] = {X 14.6392, Y 34.4030, Z -3.0000, A 0.000, B 0.000, C 0.000 }
gfCNCPoint2[24381] = {X 10.6875, Y 35.0226, Z -3.0000, A 0.000, B 0.000, C 0.000 }
gfCNCPoint2[24382] = {X 14.7702, Y 36.3185, Z -3.0000, A 0.000, B 0.000, C 0.000 }
gfCNCPoint2[24383] = {X 14.6337, Y 34.3232, Z -3.0000, A 0.000, B 0.000, C 0.000 }
gfCNCPoint2[24384] = {X 12.2421, Y 34.4753, Z -3.0000, A 0.000, B 0.000, C 0.000 }
gfCNCPoint2[24385] = {X 9.8492, Y 34.6046, Z -3.0000, A 0.000, B 0.000, C 0.000 }
gfCNCPoint2[24386] = {X 8.5934, Y 34.7137, Z -3.0000, A 0.000, B 0.000, C 0.000 }
gfCNCPoint2[24387] = {X 7.3605, Y 34.9761, Z -3.0000, A 0.000, B 0.000, C 0.000 }
gfCNCPoint2[24388] = {X 7.2796, Y 35.1977, Z -3.0000, A 0.000, B 0.000, C 0.000 }
gfCNCPoint2[24389] = {X 7.2516, Y 35.4320, Z -3.0000, A 0.000, B 0.000, C 0.000 }
gfCNCPoint2[24390] = {X 7.3209, Y 35.9826, Z -3.0000, A 0.000, B 0.000, C 0.000 }
gfCNCPoint2[24391] = {X 7.5283, Y 36.4974, Z -3.0000, A 0.000, B 0.000, C 0.000 }
gfCNCPoint2[24392] = {X 7.8601, Y 36.9423, Z -3.0000, A 0.000, B 0.000, C 0.000 }
gfCNCPoint2[24393] = {X 8.2943, Y 37.2879, Z -3.0000, A 0.000, B 0.000, C 0.000 }
gfCNCPoint2[24394] = {X 9.1179, Y 37.7054, Z -3.0000, A 0.000, B 0.000, C 0.000 }
gfCNCPoint2[24395] = {X 9.9942, Y 37.9966, Z -3.0000, A 0.000, B 0.000, C 0.000 }
gfCNCPoint2[24396] = {X 11.3207, Y 38.2433, Z -3.0000, A 0.000, B 0.000, C 0.000 }
gfCNCPoint2[24397] = {X 12.6676, Y 38.3220, Z -3.0000, A 0.000, B 0.000, C 0.000 }
gfCNCPoint2[24398] = {X 14.0138, Y 38.2314, Z -3.0000, A 0.000, B 0.000, C 0.000 }
gfCNCPoint2[24399] = {X 15.3381, Y 37.9730, Z -3.0000, A 0.000, B 0.000, C 0.000 }
gfCNCPoint2[24400] = {X 16.6196, Y 37.5507, Z -3.0000, A 0.000, B 0.000, C 0.000 }
gfCNCPoint2[24401] = {X 18.0692, Y 36.8696, Z -3.0000, A 0.000, B 0.000, C 0.000 }
gfCNCPoint2[24402] = {X 19.4300, Y 36.0248, Z -3.0000, A 0.000, B 0.000, C 0.000 }
gfCNCPoint2[24403] = {X 19.5226, Y 35.1553, Z -3.0000, A 0.000, B 0.000, C 0.000 }
gfCNCPoint2[24404] = {X 19.8019, Y 34.3266, Z -3.0000, A 0.000, B 0.000, C 0.000 }
gfCNCPoint2[24405] = {X 20.2547, Y 33.5784, Z -3.0000, A 0.000, B 0.000, C 0.000 }
gfCNCPoint2[24406] = {X 18.1811, Y 33.9836, Z -3.0000, A 0.000, B 0.000, C 0.000 }
gfCNCPoint2[24407] = {X 16.0816, Y 34.2200, Z -3.0000, A 0.000, B 0.000, C 0.000 }
gfCNCPoint2[24408] = {X 15.3577, Y 34.2726, Z -3.0000, A 0.000, B 0.000, C 0.000 }
gfCNCPoint2[24409] = {X 14.6337, Y 34.3232, Z -3.0000, A 0.000, B 0.000, C 0.000 }
gfCNCPoint2[24410] = {X 14.7702, Y 36.3185, Z -3.0000, A 0.000, B 0.000, C 0.000 }
gfCNCPoint2[24411] = {X 14.7702, Y 36.3185, Z 0.0000, A 0.000, B 0.000, C 0.000 }
gfCNCPoint2[24412] = {X 14.7702, Y 36.3185, Z 11.0000, A 0.000, B 0.000, C 0.000 }
gfCNCPoint2[24413] = {X 15.0748, Y 19.4916, Z 11.0000, A 0.000, B 0.000, C 0.000 }
gfCNCPoint2[24414] = {X 15.0748, Y 19.4916, Z 0.8333, A 0.000, B 0.000, C 0.000 }
gfCNCPoint2[24415] = {X 14.5039, Y 19.3624, Z 0.6765, A 0.000, B 0.000, C 0.000 }
gfCNCPoint2[24416] = {X 13.3045, Y 19.2487, Z 0.3537, A 0.000, B 0.000, C 0.000 }
gfCNCPoint2[24417] = {X 12.0998, Y 19.2661, Z 0.0308, A 0.000, B 0.000, C 0.000 }
gfCNCPoint2[24418] = {X 11.2937, Y 19.3818, Z -0.1874, A 0.000, B 0.000, C 0.000 }
gfCNCPoint2[24419] = {X 10.6070, Y 19.4898, Z -0.3736, A 0.000, B 0.000, C 0.000 }
gfCNCPoint2[24420] = {X 9.8988, Y 19.6129, Z -0.5662, A 0.000, B 0.000, C 0.000 }
gfCNCPoint2[24421] = {X 8.6153, Y 20.0589, Z -0.9303, A 0.000, B 0.000, C 0.000 }
gfCNCPoint2[24422] = {X 7.9833, Y 20.4014, Z -1.1229, A 0.000, B 0.000, C 0.000 }
gfCNCPoint2[24423] = {X 7.9274, Y 20.9131, Z -1.2608, A 0.000, B 0.000, C 0.000 }
gfCNCPoint2[24424] = {X 7.4488, Y 22.1330, Z -1.6120, A 0.000, B 0.000, C 0.000 }
gfCNCPoint2[24425] = {X 7.1420, Y 22.5462, Z -1.7499, A 0.000, B 0.000, C 0.000 }
gfCNCPoint2[24426] = {X 8.6590, Y 22.3492, Z -2.1597, A 0.000, B 0.000, C 0.000 }
gfCNCPoint2[24427] = {X 8.9965, Y 22.3202, Z -2.2505, A 0.000, B 0.000, C 0.000 }
gfCNCPoint2[24428] = {X 10.5268, Y 22.2558, Z -2.6609, A 0.000, B 0.000, C 0.000 }
gfCNCPoint2[24429] = {X 11.1591, Y 22.2322, Z -2.8305, A 0.000, B 0.000, C 0.000 }
gfCNCPoint2[24430] = {X 11.7911, Y 22.2030, Z -3.0000, A 0.000, B 0.000, C 0.000 }
gfCNCPoint2[24431] = {X 14.1196, Y 22.0771, Z -3.0000, A 0.000, B 0.000, C 0.000 }
gfCNCPoint2[24432] = {X 16.4457, Y 21.9141, Z -3.0000, A 0.000, B 0.000, C 0.000 }
gfCNCPoint2[24433] = {X 17.0566, Y 21.8302, Z -3.0000, A 0.000, B 0.000, C 0.000 }
gfCNCPoint2[24434] = {X 17.6535, Y 21.6756, Z -3.0000, A 0.000, B 0.000, C 0.000 }
gfCNCPoint2[24435] = {X 17.6750, Y 21.2161, Z -3.0000, A 0.000, B 0.000, C 0.000 }
gfCNCPoint2[24436] = {X 17.5250, Y 20.7812, Z -3.0000, A 0.000, B 0.000, C 0.000 }
gfCNCPoint2[24437] = {X 17.2247, Y 20.4327, Z -3.0000, A 0.000, B 0.000, C 0.000 }
gfCNCPoint2[24438] = {X 16.3055, Y 19.8922, Z -3.0000, A 0.000, B 0.000, C 0.000 }
gfCNCPoint2[24439] = {X 15.2982, Y 19.5421, Z -3.0000, A 0.000, B 0.000, C 0.000 }
gfCNCPoint2[24440] = {X 13.9732, Y 19.3260, Z -3.0000, A 0.000, B 0.000, C 0.000 }
gfCNCPoint2[24441] = {X 12.6317, Y 19.2723, Z -3.0000, A 0.000, B 0.000, C 0.000 }
gfCNCPoint2[24442] = {X 11.2937, Y 19.3818, Z -3.0000, A 0.000, B 0.000, C 0.000 }
gfCNCPoint2[24443] = {X 10.6070, Y 19.4898, Z -3.0000, A 0.000, B 0.000, C 0.000 }
gfCNCPoint2[24444] = {X 9.2581, Y 19.8389, Z -3.0000, A 0.000, B 0.000, C 0.000 }
gfCNCPoint2[24445] = {X 7.9833, Y 20.4014, Z -3.0000, A 0.000, B 0.000, C 0.000 }
gfCNCPoint2[24446] = {X 7.8313, Y 21.1624, Z -3.0000, A 0.000, B 0.000, C 0.000 }
gfCNCPoint2[24447] = {X 7.5479, Y 21.8848, Z -3.0000, A 0.000, B 0.000, C 0.000 }
gfCNCPoint2[24448] = {X 7.1420, Y 22.5462, Z -3.0000, A 0.000, B 0.000, C 0.000 }
gfCNCPoint2[24449] = {X 8.8312, Y 22.3641, Z -3.0000, A 0.000, B 0.000, C 0.000 }
gfCNCPoint2[24450] = {X 10.5268, Y 22.2558, Z -3.0000, A 0.000, B 0.000, C 0.000 }
gfCNCPoint2[24451] = {X 11.1590, Y 22.2308, Z -3.0000, A 0.000, B 0.000, C 0.000 }
gfCNCPoint2[24452] = {X 11.7911, Y 22.2030, Z -3.0000, A 0.000, B 0.000, C 0.000 }
gfCNCPoint2[24453] = {X 7.7982, Y 22.1181, Z -3.0000, A 0.000, B 0.000, C 0.000 }
gfCNCPoint2[24454] = {X 11.7948, Y 22.2830, Z -3.0000, A 0.000, B 0.000, C 0.000 }
gfCNCPoint2[24455] = {X 14.1245, Y 22.1570, Z -3.0000, A 0.000, B 0.000, C 0.000 }
gfCNCPoint2[24456] = {X 16.4519, Y 21.9938, Z -3.0000, A 0.000, B 0.000, C 0.000 }
gfCNCPoint2[24457] = {X 17.0937, Y 21.9043, Z -3.0000, A 0.000, B 0.000, C 0.000 }
gfCNCPoint2[24458] = {X 17.7199, Y 21.7380, Z -3.0000, A 0.000, B 0.000, C 0.000 }
gfCNCPoint2[24459] = {X 17.7581, Y 21.2340, Z -3.0000, A 0.000, B 0.000, C 0.000 }
gfCNCPoint2[24460] = {X 17.6012, Y 20.7535, Z -3.0000, A 0.000, B 0.000, C 0.000 }
gfCNCPoint2[24461] = {X 17.2731, Y 20.3690, Z -3.0000, A 0.000, B 0.000, C 0.000 }
gfCNCPoint2[24462] = {X 16.3395, Y 19.8198, Z -3.0000, A 0.000, B 0.000, C 0.000 }
gfCNCPoint2[24463] = {X 15.3164, Y 19.4642, Z -3.0000, A 0.000, B 0.000, C 0.000 }
gfCNCPoint2[24464] = {X 13.9814, Y 19.2464, Z -3.0000, A 0.000, B 0.000, C 0.000 }
gfCNCPoint2[24465] = {X 12.6299, Y 19.1923, Z -3.0000, A 0.000, B 0.000, C 0.000 }
gfCNCPoint2[24466] = {X 11.2818, Y 19.3027, Z -3.0000, A 0.000, B 0.000, C 0.000 }
gfCNCPoint2[24467] = {X 10.5939, Y 19.4108, Z -3.0000, A 0.000, B 0.000, C 0.000 }
gfCNCPoint2[24468] = {X 9.2122, Y 19.7702, Z -3.0000, A 0.000, B 0.000, C 0.000 }
gfCNCPoint2[24469] = {X 7.9081, Y 20.3513, Z -3.0000, A 0.000, B 0.000, C 0.000 }
gfCNCPoint2[24470] = {X 7.7440, Y 21.1750, Z -3.0000, A 0.000, B 0.000, C 0.000 }
gfCNCPoint2[24471] = {X 7.4236, Y 21.9514, Z -3.0000, A 0.000, B 0.000, C 0.000 }
gfCNCPoint2[24472] = {X 6.9591, Y 22.6511, Z -3.0000, A 0.000, B 0.000, C 0.000 }
gfCNCPoint2[24473] = {X 8.7400, Y 22.4524, Z -3.0000, A 0.000, B 0.000, C 0.000 }
gfCNCPoint2[24474] = {X 10.5282, Y 22.3358, Z -3.0000, A 0.000, B 0.000, C 0.000 }
gfCNCPoint2[24475] = {X 11.1616, Y 22.3108, Z -3.0000, A 0.000, B 0.000, C 0.000 }
gfCNCPoint2[24476] = {X 11.7948, Y 22.2830, Z -3.0000, A 0.000, B 0.000, C 0.000 }
gfCNCPoint2[24477] = {X 15.7593, Y 21.7513, Z -3.0000, A 0.000, B 0.000, C 0.000 }
gfCNCPoint2[24478] = {X 7.8019, Y 22.1980, Z -3.0000, A 0.000, B 0.000, C 0.000 }
gfCNCPoint2[24479] = {X 11.7985, Y 22.3629, Z -3.0000, A 0.000, B 0.000, C 0.000 }
gfCNCPoint2[24480] = {X 14.1295, Y 22.2368, Z -3.0000, A 0.000, B 0.000, C 0.000 }
gfCNCPoint2[24481] = {X 16.4582, Y 22.0736, Z -3.0000, A 0.000, B 0.000, C 0.000 }
gfCNCPoint2[24482] = {X 17.1301, Y 21.9786, Z -3.0000, A 0.000, B 0.000, C 0.000 }
gfCNCPoint2[24483] = {X 17.7849, Y 21.8006, Z -3.0000, A 0.000, B 0.000, C 0.000 }
gfCNCPoint2[24484] = {X 17.8406, Y 21.2523, Z -3.0000, A 0.000, B 0.000, C 0.000 }
gfCNCPoint2[24485] = {X 17.6775, Y 20.7260, Z -3.0000, A 0.000, B 0.000, C 0.000 }
gfCNCPoint2[24486] = {X 17.3215, Y 20.3053, Z -3.0000, A 0.000, B 0.000, C 0.000 }
gfCNCPoint2[24487] = {X 16.3736, Y 19.7474, Z -3.0000, A 0.000, B 0.000, C 0.000 }
gfCNCPoint2[24488] = {X 15.3346, Y 19.3863, Z -3.0000, A 0.000, B 0.000, C 0.000 }
gfCNCPoint2[24489] = {X 13.9897, Y 19.1668, Z -3.0000, A 0.000, B 0.000, C 0.000 }
gfCNCPoint2[24490] = {X 12.6280, Y 19.1123, Z -3.0000, A 0.000, B 0.000, C 0.000 }
gfCNCPoint2[24491] = {X 11.2699, Y 19.2236, Z -3.0000, A 0.000, B 0.000, C 0.000 }
gfCNCPoint2[24492] = {X 10.5809, Y 19.3319, Z -3.0000, A 0.000, B 0.000, C 0.000 }
gfCNCPoint2[24493] = {X 9.6302, Y 19.5522, Z -3.0000, A 0.000, B 0.000, C 0.000 }
gfCNCPoint2[24494] = {X 8.7100, Y 19.8770, Z -3.0000, A 0.000, B 0.000, C 0.000 }
gfCNCPoint2[24495] = {X 7.8316, Y 20.3021, Z -3.0000, A 0.000, B 0.000, C 0.000 }
gfCNCPoint2[24496] = {X 7.8285, Y 20.3434, Z -3.0000, A 0.000, B 0.000, C 0.000 }
gfCNCPoint2[24497] = {X 7.6468, Y 21.2182, Z -3.0000, A 0.000, B 0.000, C 0.000 }
gfCNCPoint2[24498] = {X 7.2857, Y 22.0356, Z -3.0000, A 0.000, B 0.000, C 0.000 }
gfCNCPoint2[24499] = {X 6.7613, Y 22.7591, Z -3.0000, A 0.000, B 0.000, C 0.000 }
gfCNCPoint2[24500] = {X 8.6423, Y 22.5415, Z -3.0000, A 0.000, B 0.000, C 0.000 }
gfCNCPoint2[24501] = {X 10.5316, Y 22.4158, Z -3.0000, A 0.000, B 0.000, C 0.000 }
gfCNCPoint2[24502] = {X 11.1651, Y 22.3907, Z -3.0000, A 0.000, B 0.000, C 0.000 }
gfCNCPoint2[24503] = {X 11.7985, Y 22.3629, Z -3.0000, A 0.000, B 0.000, C 0.000 }
gfCNCPoint2[24504] = {X 15.7630, Y 21.8312, Z -3.0000, A 0.000, B 0.000, C 0.000 }
gfCNCPoint2[24505] = {X 7.8056, Y 22.2780, Z -3.0000, A 0.000, B 0.000, C 0.000 }
gfCNCPoint2[24506] = {X 11.8022, Y 22.4428, Z -3.0000, A 0.000, B 0.000, C 0.000 }
gfCNCPoint2[24507] = {X 14.1345, Y 22.3167, Z -3.0000, A 0.000, B 0.000, C 0.000 }
gfCNCPoint2[24508] = {X 16.4644, Y 22.1533, Z -3.0000, A 0.000, B 0.000, C 0.000 }
gfCNCPoint2[24509] = {X 17.1658, Y 22.0529, Z -3.0000, A 0.000, B 0.000, C 0.000 }
gfCNCPoint2[24510] = {X 17.8485, Y 21.8633, Z -3.0000, A 0.000, B 0.000, C 0.000 }
gfCNCPoint2[24511] = {X 17.9271, Y 21.4212, Z -3.0000, A 0.000, B 0.000, C 0.000 }
gfCNCPoint2[24512] = {X 17.8677, Y 20.9761, Z -3.0000, A 0.000, B 0.000, C 0.000 }
gfCNCPoint2[24513] = {X 17.6759, Y 20.5701, Z -3.0000, A 0.000, B 0.000, C 0.000 }
gfCNCPoint2[24514] = {X 17.3699, Y 20.2415, Z -3.0000, A 0.000, B 0.000, C 0.000 }
gfCNCPoint2[24515] = {X 16.4076, Y 19.6750, Z -3.0000, A 0.000, B 0.000, C 0.000 }
gfCNCPoint2[24516] = {X 15.3527, Y 19.3084, Z -3.0000, A 0.000, B 0.000, C 0.000 }
gfCNCPoint2[24517] = {X 13.9979, Y 19.0872, Z -3.0000, A 0.000, B 0.000, C 0.000 }
gfCNCPoint2[24518] = {X 12.6262, Y 19.0323, Z -3.0000, A 0.000, B 0.000, C 0.000 }
gfCNCPoint2[24519] = {X 11.2580, Y 19.1445, Z -3.0000, A 0.000, B 0.000, C 0.000 }
gfCNCPoint2[24520] = {X 10.5678, Y 19.2530, Z -3.0000, A 0.000, B 0.000, C 0.000 }
gfCNCPoint2[24521] = {X 9.5944, Y 19.4794, Z -3.0000, A 0.000, B 0.000, C 0.000 }
gfCNCPoint2[24522] = {X 8.6527, Y 19.8142, Z -3.0000, A 0.000, B 0.000, C 0.000 }
gfCNCPoint2[24523] = {X 7.7550, Y 20.2533, Z -3.0000, A 0.000, B 0.000, C 0.000 }
gfCNCPoint2[24524] = {X 7.7493, Y 20.3320, Z -3.0000, A 0.000, B 0.000, C 0.000 }
gfCNCPoint2[24525] = {X 7.5474, Y 21.2639, Z -3.0000, A 0.000, B 0.000, C 0.000 }
gfCNCPoint2[24526] = {X 7.1387, Y 22.1253, Z -3.0000, A 0.000, B 0.000, C 0.000 }
gfCNCPoint2[24527] = {X 6.5445, Y 22.8711, Z -3.0000, A 0.000, B 0.000, C 0.000 }
gfCNCPoint2[24528] = {X 8.5349, Y 22.6317, Z -3.0000, A 0.000, B 0.000, C 0.000 }
gfCNCPoint2[24529] = {X 10.5350, Y 22.4957, Z -3.0000, A 0.000, B 0.000, C 0.000 }
gfCNCPoint2[24530] = {X 11.1686, Y 22.4706, Z -3.0000, A 0.000, B 0.000, C 0.000 }
gfCNCPoint2[24531] = {X 11.8022, Y 22.4428, Z -3.0000, A 0.000, B 0.000, C 0.000 }
gfCNCPoint2[24532] = {X 15.7667, Y 21.9111, Z -3.0000, A 0.000, B 0.000, C 0.000 }
gfCNCPoint2[24533] = {X 7.8093, Y 22.3579, Z -3.0000, A 0.000, B 0.000, C 0.000 }
gfCNCPoint2[24534] = {X 11.8059, Y 22.5227, Z -3.0000, A 0.000, B 0.000, C 0.000 }
gfCNCPoint2[24535] = {X 14.1394, Y 22.3965, Z -3.0000, A 0.000, B 0.000, C 0.000 }
gfCNCPoint2[24536] = {X 16.4706, Y 22.2331, Z -3.0000, A 0.000, B 0.000, C 0.000 }
gfCNCPoint2[24537] = {X 17.2010, Y 22.1272, Z -3.0000, A 0.000, B 0.000, C 0.000 }
gfCNCPoint2[24538] = {X 17.9111, Y 21.9261, Z -3.0000, A 0.000, B 0.000, C 0.000 }
gfCNCPoint2[24539] = {X 18.0062, Y 21.4519, Z -3.0000, A 0.000, B 0.000, C 0.000 }
gfCNCPoint2[24540] = {X 17.9496, Y 20.9716, Z -3.0000, A 0.000, B 0.000, C 0.000 }
gfCNCPoint2[24541] = {X 17.7470, Y 20.5325, Z -3.0000, A 0.000, B 0.000, C 0.000 }
gfCNCPoint2[24542] = {X 17.4182, Y 20.1778, Z -3.0000, A 0.000, B 0.000, C 0.000 }
gfCNCPoint2[24543] = {X 16.4416, Y 19.6026, Z -3.0000, A 0.000, B 0.000, C 0.000 }
gfCNCPoint2[24544] = {X 15.3709, Y 19.2305, Z -3.0000, A 0.000, B 0.000, C 0.000 }
gfCNCPoint2[24545] = {X 14.0061, Y 19.0077, Z -3.0000, A 0.000, B 0.000, C 0.000 }
gfCNCPoint2[24546] = {X 12.6243, Y 18.9523, Z -3.0000, A 0.000, B 0.000, C 0.000 }
gfCNCPoint2[24547] = {X 11.2461, Y 19.0654, Z -3.0000, A 0.000, B 0.000, C 0.000 }
gfCNCPoint2[24548] = {X 10.5548, Y 19.1740, Z -3.0000, A 0.000, B 0.000, C 0.000 }
gfCNCPoint2[24549] = {X 9.5585, Y 19.4065, Z -3.0000, A 0.000, B 0.000, C 0.000 }
gfCNCPoint2[24550] = {X 8.5954, Y 19.7516, Z -3.0000, A 0.000, B 0.000, C 0.000 }
gfCNCPoint2[24551] = {X 7.6783, Y 20.2047, Z -3.0000, A 0.000, B 0.000, C 0.000 }
gfCNCPoint2[24552] = {X 7.6696, Y 20.3251, Z -3.0000, A 0.000, B 0.000, C 0.000 }
gfCNCPoint2[24553] = {X 7.5231, Y 21.0762, Z -3.0000, A 0.000, B 0.000, C 0.000 }
gfCNCPoint2[24554] = {X 7.2389, Y 21.7867, Z -3.0000, A 0.000, B 0.000, C 0.000 }
gfCNCPoint2[24555] = {X 6.8271, Y 22.4316, Z -3.0000, A 0.000, B 0.000, C 0.000 }
gfCNCPoint2[24556] = {X 6.3021, Y 22.9883, Z -3.0000, A 0.000, B 0.000, C 0.000 }
gfCNCPoint2[24557] = {X 8.4146, Y 22.7236, Z -3.0000, A 0.000, B 0.000, C 0.000 }
gfCNCPoint2[24558] = {X 10.5383, Y 22.5756, Z -3.0000, A 0.000, B 0.000, C 0.000 }
gfCNCPoint2[24559] = {X 11.1722, Y 22.5505, Z -3.0000, A 0.000, B 0.000, C 0.000 }
gfCNCPoint2[24560] = {X 11.8059, Y 22.5227, Z -3.0000, A 0.000, B 0.000, C 0.000 }
gfCNCPoint2[24561] = {X 15.7704, Y 21.9910, Z -3.0000, A 0.000, B 0.000, C 0.000 }
gfCNCPoint2[24562] = {X 11.7345, Y 22.6061, Z -3.0000, A 0.000, B 0.000, C 0.000 }
gfCNCPoint2[24563] = {X 11.8095, Y 22.6026, Z -3.0000, A 0.000, B 0.000, C 0.000 }
gfCNCPoint2[24564] = {X 14.1444, Y 22.4764, Z -3.0000, A 0.000, B 0.000, C 0.000 }
gfCNCPoint2[24565] = {X 16.4769, Y 22.3128, Z -3.0000, A 0.000, B 0.000, C 0.000 }
gfCNCPoint2[24566] = {X 17.2357, Y 22.2016, Z -3.0000, A 0.000, B 0.000, C 0.000 }
gfCNCPoint2[24567] = {X 17.9726, Y 21.9890, Z -3.0000, A 0.000, B 0.000, C 0.000 }
gfCNCPoint2[24568] = {X 18.0847, Y 21.4829, Z -3.0000, A 0.000, B 0.000, C 0.000 }
gfCNCPoint2[24569] = {X 18.0314, Y 20.9673, Z -3.0000, A 0.000, B 0.000, C 0.000 }
gfCNCPoint2[24570] = {X 17.8181, Y 20.4949, Z -3.0000, A 0.000, B 0.000, C 0.000 }
gfCNCPoint2[24571] = {X 17.4665, Y 20.1140, Z -3.0000, A 0.000, B 0.000, C 0.000 }
gfCNCPoint2[24572] = {X 16.4755, Y 19.5301, Z -3.0000, A 0.000, B 0.000, C 0.000 }
gfCNCPoint2[24573] = {X 15.3891, Y 19.1526, Z -3.0000, A 0.000, B 0.000, C 0.000 }
gfCNCPoint2[24574] = {X 14.0143, Y 18.9281, Z -3.0000, A 0.000, B 0.000, C 0.000 }
gfCNCPoint2[24575] = {X 12.6225, Y 18.8724, Z -3.0000, A 0.000, B 0.000, C 0.000 }
gfCNCPoint2[24576] = {X 11.2342, Y 18.9863, Z -3.0000, A 0.000, B 0.000, C 0.000 }
gfCNCPoint2[24577] = {X 10.5417, Y 19.0951, Z -3.0000, A 0.000, B 0.000, C 0.000 }
gfCNCPoint2[24578] = {X 9.5226, Y 19.3337, Z -3.0000, A 0.000, B 0.000, C 0.000 }
gfCNCPoint2[24579] = {X 8.5381, Y 19.6891, Z -3.0000, A 0.000, B 0.000, C 0.000 }
gfCNCPoint2[24580] = {X 7.6015, Y 20.1564, Z -3.0000, A 0.000, B 0.000, C 0.000 }
gfCNCPoint2[24581] = {X 7.5898, Y 20.3183, Z -3.0000, A 0.000, B 0.000, C 0.000 }
gfCNCPoint2[24582] = {X 7.4461, Y 21.0543, Z -3.0000, A 0.000, B 0.000, C 0.000 }
gfCNCPoint2[24583] = {X 7.1675, Y 21.7506, Z -3.0000, A 0.000, B 0.000, C 0.000 }
gfCNCPoint2[24584] = {X 6.7639, Y 22.3826, Z -3.0000, A 0.000, B 0.000, C 0.000 }
gfCNCPoint2[24585] = {X 6.2493, Y 22.9282, Z -3.0000, A 0.000, B 0.000, C 0.000 }
gfCNCPoint2[24586] = {X 6.2078, Y 22.9642, Z -3.0000, A 0.000, B 0.000, C 0.000 }
gfCNCPoint2[24587] = {X 6.1658, Y 22.9996, Z -3.0000, A 0.000, B 0.000, C 0.000 }
gfCNCPoint2[24588] = {X 6.1506, Y 23.0928, Z -3.0000, A 0.000, B 0.000, C 0.000 }
gfCNCPoint2[24589] = {X 6.2324, Y 23.0800, Z -3.0000, A 0.000, B 0.000, C 0.000 }
gfCNCPoint2[24590] = {X 6.3143, Y 23.0674, Z -3.0000, A 0.000, B 0.000, C 0.000 }
gfCNCPoint2[24591] = {X 8.4223, Y 22.8032, Z -3.0000, A 0.000, B 0.000, C 0.000 }
gfCNCPoint2[24592] = {X 10.5417, Y 22.6555, Z -3.0000, A 0.000, B 0.000, C 0.000 }
gfCNCPoint2[24593] = {X 11.1757, Y 22.6305, Z -3.0000, A 0.000, B 0.000, C 0.000 }
gfCNCPoint2[24594] = {X 11.8095, Y 22.6026, Z -3.0000, A 0.000, B 0.000, C 0.000 }
gfCNCPoint2[24595] = {X 11.7175, Y 20.6047, Z -3.0000, A 0.000, B 0.000, C 0.000 }
gfCNCPoint2[24596] = {X 11.7175, Y 20.6047, Z 0.0000, A 0.000, B 0.000, C 0.000 }
gfCNCPoint2[24597] = {X 11.7175, Y 20.6047, Z 11.0000, A 0.000, B 0.000, C 0.000 }
gfCNCPoint2[24598] = {X 15.0757, Y 19.4921, Z 11.0000, A 0.000, B 0.000, C 0.000 }
gfCNCPoint2[24599] = {X 15.0757, Y 19.4921, Z 0.0000, A 0.000, B 0.000, C 0.000 }
gfCNCPoint2[24600] = {X 14.5039, Y 19.3627, Z -0.1571, A 0.000, B 0.000, C 0.000 }
gfCNCPoint2[24601] = {X 13.3045, Y 19.2491, Z -0.4799, A 0.000, B 0.000, C 0.000 }
gfCNCPoint2[24602] = {X 12.0998, Y 19.2665, Z -0.8027, A 0.000, B 0.000, C 0.000 }
gfCNCPoint2[24603] = {X 11.2937, Y 19.3821, Z -1.0209, A 0.000, B 0.000, C 0.000 }
gfCNCPoint2[24604] = {X 10.6070, Y 19.4901, Z -1.2072, A 0.000, B 0.000, C 0.000 }
gfCNCPoint2[24605] = {X 9.8989, Y 19.6132, Z -1.3998, A 0.000, B 0.000, C 0.000 }
gfCNCPoint2[24606] = {X 8.6151, Y 20.0593, Z -1.7639, A 0.000, B 0.000, C 0.000 }
gfCNCPoint2[24607] = {X 7.9833, Y 20.4018, Z -1.9565, A 0.000, B 0.000, C 0.000 }
gfCNCPoint2[24608] = {X 7.9273, Y 20.9134, Z -2.0944, A 0.000, B 0.000, C 0.000 }
gfCNCPoint2[24609] = {X 7.4491, Y 22.1326, Z -2.4453, A 0.000, B 0.000, C 0.000 }
gfCNCPoint2[24610] = {X 7.1423, Y 22.5459, Z -2.5832, A 0.000, B 0.000, C 0.000 }
gfCNCPoint2[24611] = {X 8.6593, Y 22.3488, Z -2.9931, A 0.000, B 0.000, C 0.000 }
gfCNCPoint2[24612] = {X 8.9965, Y 22.3199, Z -3.0838, A 0.000, B 0.000, C 0.000 }
gfCNCPoint2[24613] = {X 10.5268, Y 22.2555, Z -3.4942, A 0.000, B 0.000, C 0.000 }
gfCNCPoint2[24614] = {X 11.1591, Y 22.2318, Z -3.6638, A 0.000, B 0.000, C 0.000 }
gfCNCPoint2[24615] = {X 11.7912, Y 22.2027, Z -3.8333, A 0.000, B 0.000, C 0.000 }
gfCNCPoint2[24616] = {X 14.1195, Y 22.0768, Z -3.8333, A 0.000, B 0.000, C 0.000 }
gfCNCPoint2[24617] = {X 16.4456, Y 21.9137, Z -3.8333, A 0.000, B 0.000, C 0.000 }
gfCNCPoint2[24618] = {X 17.0564, Y 21.8299, Z -3.8333, A 0.000, B 0.000, C 0.000 }
gfCNCPoint2[24619] = {X 17.6532, Y 21.6754, Z -3.8333, A 0.000, B 0.000, C 0.000 }
gfCNCPoint2[24620] = {X 17.6747, Y 21.2161, Z -3.8333, A 0.000, B 0.000, C 0.000 }
gfCNCPoint2[24621] = {X 17.5247, Y 20.7814, Z -3.8333, A 0.000, B 0.000, C 0.000 }
gfCNCPoint2[24622] = {X 17.2247, Y 20.4330, Z -3.8333, A 0.000, B 0.000, C 0.000 }
gfCNCPoint2[24623] = {X 16.3055, Y 19.8925, Z -3.8333, A 0.000, B 0.000, C 0.000 }
gfCNCPoint2[24624] = {X 15.2982, Y 19.5425, Z -3.8333, A 0.000, B 0.000, C 0.000 }
gfCNCPoint2[24625] = {X 13.9732, Y 19.3263, Z -3.8333, A 0.000, B 0.000, C 0.000 }
gfCNCPoint2[24626] = {X 12.6317, Y 19.2726, Z -3.8333, A 0.000, B 0.000, C 0.000 }
gfCNCPoint2[24627] = {X 11.2937, Y 19.3821, Z -3.8333, A 0.000, B 0.000, C 0.000 }
gfCNCPoint2[24628] = {X 10.6070, Y 19.4901, Z -3.8333, A 0.000, B 0.000, C 0.000 }
gfCNCPoint2[24629] = {X 9.2581, Y 19.8392, Z -3.8333, A 0.000, B 0.000, C 0.000 }
gfCNCPoint2[24630] = {X 7.9833, Y 20.4018, Z -3.8333, A 0.000, B 0.000, C 0.000 }
gfCNCPoint2[24631] = {X 7.8312, Y 21.1625, Z -3.8333, A 0.000, B 0.000, C 0.000 }
gfCNCPoint2[24632] = {X 7.5480, Y 21.8847, Z -3.8333, A 0.000, B 0.000, C 0.000 }
gfCNCPoint2[24633] = {X 7.1423, Y 22.5459, Z -3.8333, A 0.000, B 0.000, C 0.000 }
gfCNCPoint2[24634] = {X 8.8313, Y 22.3638, Z -3.8333, A 0.000, B 0.000, C 0.000 }
gfCNCPoint2[24635] = {X 10.5268, Y 22.2555, Z -3.8333, A 0.000, B 0.000, C 0.000 }
gfCNCPoint2[24636] = {X 11.1590, Y 22.2305, Z -3.8333, A 0.000, B 0.000, C 0.000 }
gfCNCPoint2[24637] = {X 11.7912, Y 22.2027, Z -3.8333, A 0.000, B 0.000, C 0.000 }
gfCNCPoint2[24638] = {X 7.7983, Y 22.1178, Z -3.8333, A 0.000, B 0.000, C 0.000 }
gfCNCPoint2[24639] = {X 11.7949, Y 22.2826, Z -3.8333, A 0.000, B 0.000, C 0.000 }
gfCNCPoint2[24640] = {X 14.1245, Y 22.1566, Z -3.8333, A 0.000, B 0.000, C 0.000 }
gfCNCPoint2[24641] = {X 16.4518, Y 21.9935, Z -3.8333, A 0.000, B 0.000, C 0.000 }
gfCNCPoint2[24642] = {X 17.0935, Y 21.9041, Z -3.8333, A 0.000, B 0.000, C 0.000 }
gfCNCPoint2[24643] = {X 17.7197, Y 21.7378, Z -3.8333, A 0.000, B 0.000, C 0.000 }
gfCNCPoint2[24644] = {X 17.7577, Y 21.2340, Z -3.8333, A 0.000, B 0.000, C 0.000 }
gfCNCPoint2[24645] = {X 17.6010, Y 20.7537, Z -3.8333, A 0.000, B 0.000, C 0.000 }
gfCNCPoint2[24646] = {X 17.2731, Y 20.3693, Z -3.8333, A 0.000, B 0.000, C 0.000 }
gfCNCPoint2[24647] = {X 16.3395, Y 19.8201, Z -3.8333, A 0.000, B 0.000, C 0.000 }
gfCNCPoint2[24648] = {X 15.3164, Y 19.4645, Z -3.8333, A 0.000, B 0.000, C 0.000 }
gfCNCPoint2[24649] = {X 13.9814, Y 19.2467, Z -3.8333, A 0.000, B 0.000, C 0.000 }
gfCNCPoint2[24650] = {X 12.6299, Y 19.1926, Z -3.8333, A 0.000, B 0.000, C 0.000 }
gfCNCPoint2[24651] = {X 11.2818, Y 19.3030, Z -3.8333, A 0.000, B 0.000, C 0.000 }
gfCNCPoint2[24652] = {X 10.5939, Y 19.4112, Z -3.8333, A 0.000, B 0.000, C 0.000 }
gfCNCPoint2[24653] = {X 9.2122, Y 19.7705, Z -3.8333, A 0.000, B 0.000, C 0.000 }
gfCNCPoint2[24654] = {X 7.9081, Y 20.3517, Z -3.8333, A 0.000, B 0.000, C 0.000 }
gfCNCPoint2[24655] = {X 7.7440, Y 21.1751, Z -3.8333, A 0.000, B 0.000, C 0.000 }
gfCNCPoint2[24656] = {X 7.4237, Y 21.9512, Z -3.8333, A 0.000, B 0.000, C 0.000 }
gfCNCPoint2[24657] = {X 6.9593, Y 22.6508, Z -3.8333, A 0.000, B 0.000, C 0.000 }
gfCNCPoint2[24658] = {X 8.7402, Y 22.4520, Z -3.8333, A 0.000, B 0.000, C 0.000 }
gfCNCPoint2[24659] = {X 10.5282, Y 22.3355, Z -3.8333, A 0.000, B 0.000, C 0.000 }
gfCNCPoint2[24660] = {X 11.1616, Y 22.3104, Z -3.8333, A 0.000, B 0.000, C 0.000 }
gfCNCPoint2[24661] = {X 11.7949, Y 22.2826, Z -3.8333, A 0.000, B 0.000, C 0.000 }
gfCNCPoint2[24662] = {X 15.7594, Y 21.7510, Z -3.8333, A 0.000, B 0.000, C 0.000 }
gfCNCPoint2[24663] = {X 7.8020, Y 22.1977, Z -3.8333, A 0.000, B 0.000, C 0.000 }
gfCNCPoint2[24664] = {X 11.7986, Y 22.3625, Z -3.8333, A 0.000, B 0.000, C 0.000 }
gfCNCPoint2[24665] = {X 14.1295, Y 22.2365, Z -3.8333, A 0.000, B 0.000, C 0.000 }
gfCNCPoint2[24666] = {X 16.4580, Y 22.0732, Z -3.8333, A 0.000, B 0.000, C 0.000 }
gfCNCPoint2[24667] = {X 17.1299, Y 21.9783, Z -3.8333, A 0.000, B 0.000, C 0.000 }
gfCNCPoint2[24668] = {X 17.7846, Y 21.8004, Z -3.8333, A 0.000, B 0.000, C 0.000 }
gfCNCPoint2[24669] = {X 17.8402, Y 21.2523, Z -3.8333, A 0.000, B 0.000, C 0.000 }
gfCNCPoint2[24670] = {X 17.6772, Y 20.7262, Z -3.8333, A 0.000, B 0.000, C 0.000 }
gfCNCPoint2[24671] = {X 17.3215, Y 20.3056, Z -3.8333, A 0.000, B 0.000, C 0.000 }
gfCNCPoint2[24672] = {X 16.3736, Y 19.7477, Z -3.8333, A 0.000, B 0.000, C 0.000 }
gfCNCPoint2[24673] = {X 15.3346, Y 19.3866, Z -3.8333, A 0.000, B 0.000, C 0.000 }
gfCNCPoint2[24674] = {X 13.9897, Y 19.1671, Z -3.8333, A 0.000, B 0.000, C 0.000 }
gfCNCPoint2[24675] = {X 12.6280, Y 19.1126, Z -3.8333, A 0.000, B 0.000, C 0.000 }
gfCNCPoint2[24676] = {X 11.2699, Y 19.2239, Z -3.8333, A 0.000, B 0.000, C 0.000 }
gfCNCPoint2[24677] = {X 10.5809, Y 19.3322, Z -3.8333, A 0.000, B 0.000, C 0.000 }
gfCNCPoint2[24678] = {X 9.6302, Y 19.5525, Z -3.8333, A 0.000, B 0.000, C 0.000 }
gfCNCPoint2[24679] = {X 8.7100, Y 19.8773, Z -3.8333, A 0.000, B 0.000, C 0.000 }
gfCNCPoint2[24680] = {X 7.8317, Y 20.3025, Z -3.8333, A 0.000, B 0.000, C 0.000 }
gfCNCPoint2[24681] = {X 7.8285, Y 20.3437, Z -3.8333, A 0.000, B 0.000, C 0.000 }
gfCNCPoint2[24682] = {X 7.6467, Y 21.2183, Z -3.8333, A 0.000, B 0.000, C 0.000 }
gfCNCPoint2[24683] = {X 7.2858, Y 22.0354, Z -3.8333, A 0.000, B 0.000, C 0.000 }
gfCNCPoint2[24684] = {X 6.7616, Y 22.7588, Z -3.8333, A 0.000, B 0.000, C 0.000 }
gfCNCPoint2[24685] = {X 8.6424, Y 22.5411, Z -3.8333, A 0.000, B 0.000, C 0.000 }
gfCNCPoint2[24686] = {X 10.5316, Y 22.4154, Z -3.8333, A 0.000, B 0.000, C 0.000 }
gfCNCPoint2[24687] = {X 11.1651, Y 22.3904, Z -3.8333, A 0.000, B 0.000, C 0.000 }
gfCNCPoint2[24688] = {X 11.7986, Y 22.3625, Z -3.8333, A 0.000, B 0.000, C 0.000 }
gfCNCPoint2[24689] = {X 15.7631, Y 21.8309, Z -3.8333, A 0.000, B 0.000, C 0.000 }
gfCNCPoint2[24690] = {X 7.8056, Y 22.2776, Z -3.8333, A 0.000, B 0.000, C 0.000 }
gfCNCPoint2[24691] = {X 11.8022, Y 22.4425, Z -3.8333, A 0.000, B 0.000, C 0.000 }
gfCNCPoint2[24692] = {X 14.1344, Y 22.3163, Z -3.8333, A 0.000, B 0.000, C 0.000 }
gfCNCPoint2[24693] = {X 16.4643, Y 22.1530, Z -3.8333, A 0.000, B 0.000, C 0.000 }
gfCNCPoint2[24694] = {X 17.1656, Y 22.0526, Z -3.8333, A 0.000, B 0.000, C 0.000 }
gfCNCPoint2[24695] = {X 17.8483, Y 21.8631, Z -3.8333, A 0.000, B 0.000, C 0.000 }
gfCNCPoint2[24696] = {X 17.9267, Y 21.4211, Z -3.8333, A 0.000, B 0.000, C 0.000 }
gfCNCPoint2[24697] = {X 17.8674, Y 20.9762, Z -3.8333, A 0.000, B 0.000, C 0.000 }
gfCNCPoint2[24698] = {X 17.6757, Y 20.5704, Z -3.8333, A 0.000, B 0.000, C 0.000 }
gfCNCPoint2[24699] = {X 17.3699, Y 20.2418, Z -3.8333, A 0.000, B 0.000, C 0.000 }
gfCNCPoint2[24700] = {X 16.4076, Y 19.6753, Z -3.8333, A 0.000, B 0.000, C 0.000 }
gfCNCPoint2[24701] = {X 15.3527, Y 19.3087, Z -3.8333, A 0.000, B 0.000, C 0.000 }
gfCNCPoint2[24702] = {X 13.9979, Y 19.0876, Z -3.8333, A 0.000, B 0.000, C 0.000 }
gfCNCPoint2[24703] = {X 12.6262, Y 19.0327, Z -3.8333, A 0.000, B 0.000, C 0.000 }
gfCNCPoint2[24704] = {X 11.2580, Y 19.1448, Z -3.8333, A 0.000, B 0.000, C 0.000 }
gfCNCPoint2[24705] = {X 10.5678, Y 19.2533, Z -3.8333, A 0.000, B 0.000, C 0.000 }
gfCNCPoint2[24706] = {X 9.5944, Y 19.4797, Z -3.8333, A 0.000, B 0.000, C 0.000 }
gfCNCPoint2[24707] = {X 8.6528, Y 19.8145, Z -3.8333, A 0.000, B 0.000, C 0.000 }
gfCNCPoint2[24708] = {X 7.7551, Y 20.2536, Z -3.8333, A 0.000, B 0.000, C 0.000 }
gfCNCPoint2[24709] = {X 7.7493, Y 20.3321, Z -3.8333, A 0.000, B 0.000, C 0.000 }
gfCNCPoint2[24710] = {X 7.5474, Y 21.2638, Z -3.8333, A 0.000, B 0.000, C 0.000 }
gfCNCPoint2[24711] = {X 7.1388, Y 22.1250, Z -3.8333, A 0.000, B 0.000, C 0.000 }
gfCNCPoint2[24712] = {X 6.5449, Y 22.8707, Z -3.8333, A 0.000, B 0.000, C 0.000 }
gfCNCPoint2[24713] = {X 8.5351, Y 22.6314, Z -3.8333, A 0.000, B 0.000, C 0.000 }
gfCNCPoint2[24714] = {X 10.5350, Y 22.4953, Z -3.8333, A 0.000, B 0.000, C 0.000 }
gfCNCPoint2[24715] = {X 11.1687, Y 22.4703, Z -3.8333, A 0.000, B 0.000, C 0.000 }
gfCNCPoint2[24716] = {X 11.8022, Y 22.4425, Z -3.8333, A 0.000, B 0.000, C 0.000 }
gfCNCPoint2[24717] = {X 15.7668, Y 21.9108, Z -3.8333, A 0.000, B 0.000, C 0.000 }
gfCNCPoint2[24718] = {X 7.8093, Y 22.3575, Z -3.8333, A 0.000, B 0.000, C 0.000 }
gfCNCPoint2[24719] = {X 11.8059, Y 22.5224, Z -3.8333, A 0.000, B 0.000, C 0.000 }
gfCNCPoint2[24720] = {X 14.1394, Y 22.3962, Z -3.8333, A 0.000, B 0.000, C 0.000 }
gfCNCPoint2[24721] = {X 16.4705, Y 22.2328, Z -3.8333, A 0.000, B 0.000, C 0.000 }
gfCNCPoint2[24722] = {X 17.2008, Y 22.1269, Z -3.8333, A 0.000, B 0.000, C 0.000 }
gfCNCPoint2[24723] = {X 17.9108, Y 21.9259, Z -3.8333, A 0.000, B 0.000, C 0.000 }
gfCNCPoint2[24724] = {X 18.0058, Y 21.4519, Z -3.8333, A 0.000, B 0.000, C 0.000 }
gfCNCPoint2[24725] = {X 17.9493, Y 20.9717, Z -3.8333, A 0.000, B 0.000, C 0.000 }
gfCNCPoint2[24726] = {X 17.7468, Y 20.5327, Z -3.8333, A 0.000, B 0.000, C 0.000 }
gfCNCPoint2[24727] = {X 17.4182, Y 20.1781, Z -3.8333, A 0.000, B 0.000, C 0.000 }
gfCNCPoint2[24728] = {X 16.4416, Y 19.6029, Z -3.8333, A 0.000, B 0.000, C 0.000 }
gfCNCPoint2[24729] = {X 15.3709, Y 19.2308, Z -3.8333, A 0.000, B 0.000, C 0.000 }
gfCNCPoint2[24730] = {X 14.0061, Y 19.0080, Z -3.8333, A 0.000, B 0.000, C 0.000 }
gfCNCPoint2[24731] = {X 12.6243, Y 18.9527, Z -3.8333, A 0.000, B 0.000, C 0.000 }
gfCNCPoint2[24732] = {X 11.2461, Y 19.0657, Z -3.8333, A 0.000, B 0.000, C 0.000 }
gfCNCPoint2[24733] = {X 10.5547, Y 19.1744, Z -3.8333, A 0.000, B 0.000, C 0.000 }
gfCNCPoint2[24734] = {X 9.5586, Y 19.4068, Z -3.8333, A 0.000, B 0.000, C 0.000 }
gfCNCPoint2[24735] = {X 8.5956, Y 19.7519, Z -3.8333, A 0.000, B 0.000, C 0.000 }
gfCNCPoint2[24736] = {X 7.6785, Y 20.2050, Z -3.8333, A 0.000, B 0.000, C 0.000 }
gfCNCPoint2[24737] = {X 7.6695, Y 20.3252, Z -3.8333, A 0.000, B 0.000, C 0.000 }
gfCNCPoint2[24738] = {X 7.5231, Y 21.0761, Z -3.8333, A 0.000, B 0.000, C 0.000 }
gfCNCPoint2[24739] = {X 7.2390, Y 21.7864, Z -3.8333, A 0.000, B 0.000, C 0.000 }
gfCNCPoint2[24740] = {X 6.8274, Y 22.4313, Z -3.8333, A 0.000, B 0.000, C 0.000 }
gfCNCPoint2[24741] = {X 6.3026, Y 22.9879, Z -3.8333, A 0.000, B 0.000, C 0.000 }
gfCNCPoint2[24742] = {X 8.4148, Y 22.7233, Z -3.8333, A 0.000, B 0.000, C 0.000 }
gfCNCPoint2[24743] = {X 10.5383, Y 22.5753, Z -3.8333, A 0.000, B 0.000, C 0.000 }
gfCNCPoint2[24744] = {X 11.1722, Y 22.5502, Z -3.8333, A 0.000, B 0.000, C 0.000 }
gfCNCPoint2[24745] = {X 11.8059, Y 22.5224, Z -3.8333, A 0.000, B 0.000, C 0.000 }
gfCNCPoint2[24746] = {X 15.7704, Y 21.9907, Z -3.8333, A 0.000, B 0.000, C 0.000 }
gfCNCPoint2[24747] = {X 11.7346, Y 22.6057, Z -3.8333, A 0.000, B 0.000, C 0.000 }
gfCNCPoint2[24748] = {X 11.8096, Y 22.6023, Z -3.8333, A 0.000, B 0.000, C 0.000 }
gfCNCPoint2[24749] = {X 14.1443, Y 22.4760, Z -3.8333, A 0.000, B 0.000, C 0.000 }
gfCNCPoint2[24750] = {X 16.4767, Y 22.3125, Z -3.8333, A 0.000, B 0.000, C 0.000 }
gfCNCPoint2[24751] = {X 17.2355, Y 22.2013, Z -3.8333, A 0.000, B 0.000, C 0.000 }
gfCNCPoint2[24752] = {X 17.9723, Y 21.9888, Z -3.8333, A 0.000, B 0.000, C 0.000 }
gfCNCPoint2[24753] = {X 18.0844, Y 21.4829, Z -3.8333, A 0.000, B 0.000, C 0.000 }
gfCNCPoint2[24754] = {X 18.0311, Y 20.9674, Z -3.8333, A 0.000, B 0.000, C 0.000 }
gfCNCPoint2[24755] = {X 17.8179, Y 20.4952, Z -3.8333, A 0.000, B 0.000, C 0.000 }
gfCNCPoint2[24756] = {X 17.4665, Y 20.1143, Z -3.8333, A 0.000, B 0.000, C 0.000 }
gfCNCPoint2[24757] = {X 16.4756, Y 19.5304, Z -3.8333, A 0.000, B 0.000, C 0.000 }
gfCNCPoint2[24758] = {X 15.3891, Y 19.1529, Z -3.8333, A 0.000, B 0.000, C 0.000 }
gfCNCPoint2[24759] = {X 14.0143, Y 18.9284, Z -3.8333, A 0.000, B 0.000, C 0.000 }
gfCNCPoint2[24760] = {X 12.6225, Y 18.8727, Z -3.8333, A 0.000, B 0.000, C 0.000 }
gfCNCPoint2[24761] = {X 11.2342, Y 18.9866, Z -3.8333, A 0.000, B 0.000, C 0.000 }
gfCNCPoint2[24762] = {X 10.5417, Y 19.0954, Z -3.8333, A 0.000, B 0.000, C 0.000 }
gfCNCPoint2[24763] = {X 9.5227, Y 19.3340, Z -3.8333, A 0.000, B 0.000, C 0.000 }
gfCNCPoint2[24764] = {X 8.5383, Y 19.6893, Z -3.8333, A 0.000, B 0.000, C 0.000 }
gfCNCPoint2[24765] = {X 7.6018, Y 20.1566, Z -3.8333, A 0.000, B 0.000, C 0.000 }
gfCNCPoint2[24766] = {X 7.5898, Y 20.3183, Z -3.8333, A 0.000, B 0.000, C 0.000 }
gfCNCPoint2[24767] = {X 7.4462, Y 21.0542, Z -3.8333, A 0.000, B 0.000, C 0.000 }
gfCNCPoint2[24768] = {X 7.1677, Y 21.7503, Z -3.8333, A 0.000, B 0.000, C 0.000 }
gfCNCPoint2[24769] = {X 6.7641, Y 22.3823, Z -3.8333, A 0.000, B 0.000, C 0.000 }
gfCNCPoint2[24770] = {X 6.2498, Y 22.9278, Z -3.8333, A 0.000, B 0.000, C 0.000 }
gfCNCPoint2[24771] = {X 6.2080, Y 22.9640, Z -3.8333, A 0.000, B 0.000, C 0.000 }
gfCNCPoint2[24772] = {X 6.1658, Y 22.9996, Z -3.8333, A 0.000, B 0.000, C 0.000 }
gfCNCPoint2[24773] = {X 6.1507, Y 23.0925, Z -3.8333, A 0.000, B 0.000, C 0.000 }
gfCNCPoint2[24774] = {X 6.2327, Y 23.0797, Z -3.8333, A 0.000, B 0.000, C 0.000 }
gfCNCPoint2[24775] = {X 6.3147, Y 23.0670, Z -3.8333, A 0.000, B 0.000, C 0.000 }
gfCNCPoint2[24776] = {X 8.4225, Y 22.8029, Z -3.8333, A 0.000, B 0.000, C 0.000 }
gfCNCPoint2[24777] = {X 10.5417, Y 22.6552, Z -3.8333, A 0.000, B 0.000, C 0.000 }
gfCNCPoint2[24778] = {X 11.1757, Y 22.6301, Z -3.8333, A 0.000, B 0.000, C 0.000 }
gfCNCPoint2[24779] = {X 11.8096, Y 22.6023, Z -3.8333, A 0.000, B 0.000, C 0.000 }
gfCNCPoint2[24780] = {X 11.7176, Y 20.6044, Z -3.8333, A 0.000, B 0.000, C 0.000 }
gfCNCPoint2[24781] = {X 11.7176, Y 20.6044, Z -0.8333, A 0.000, B 0.000, C 0.000 }
gfCNCPoint2[24782] = {X 11.7176, Y 20.6044, Z 11.0000, A 0.000, B 0.000, C 0.000 }
gfCNCPoint2[24783] = {X 11.7104, Y 37.8792, Z 11.0000, A 0.000, B 0.000, C 0.000 }
gfCNCPoint2[24784] = {X 11.7104, Y 37.8792, Z 0.0000, A 0.000, B 0.000, C 0.000 }
gfCNCPoint2[24785] = {X 12.4918, Y 37.9510, Z -0.2103, A 0.000, B 0.000, C 0.000 }
gfCNCPoint2[24786] = {X 14.1330, Y 37.8410, Z -0.6510, A 0.000, B 0.000, C 0.000 }
gfCNCPoint2[24787] = {X 15.7363, Y 37.4732, Z -1.0918, A 0.000, B 0.000, C 0.000 }
gfCNCPoint2[24788] = {X 16.4685, Y 37.1800, Z -1.3031, A 0.000, B 0.000, C 0.000 }
gfCNCPoint2[24789] = {X 17.3009, Y 36.8467, Z -1.5433, A 0.000, B 0.000, C 0.000 }
gfCNCPoint2[24790] = {X 18.2937, Y 36.3175, Z -1.8448, A 0.000, B 0.000, C 0.000 }
gfCNCPoint2[24791] = {X 19.0345, Y 35.8123, Z -2.0851, A 0.000, B 0.000, C 0.000 }
gfCNCPoint2[24792] = {X 19.0577, Y 35.2982, Z -2.2230, A 0.000, B 0.000, C 0.000 }
gfCNCPoint2[24793] = {X 19.2190, Y 34.6352, Z -2.4058, A 0.000, B 0.000, C 0.000 }
gfCNCPoint2[24794] = {X 19.4346, Y 34.1678, Z -2.5437, A 0.000, B 0.000, C 0.000 }
gfCNCPoint2[24795] = {X 18.1987, Y 34.4163, Z -2.8815, A 0.000, B 0.000, C 0.000 }
gfCNCPoint2[24796] = {X 17.3681, Y 34.5291, Z -3.1061, A 0.000, B 0.000, C 0.000 }
gfCNCPoint2[24797] = {X 16.1107, Y 34.6192, Z -3.4439, A 0.000, B 0.000, C 0.000 }
gfCNCPoint2[24798] = {X 15.3860, Y 34.6730, Z -3.6386, A 0.000, B 0.000, C 0.000 }
gfCNCPoint2[24799] = {X 14.6610, Y 34.7226, Z -3.8333, A 0.000, B 0.000, C 0.000 }
gfCNCPoint2[24800] = {X 12.2608, Y 34.8751, Z -3.8333, A 0.000, B 0.000, C 0.000 }
gfCNCPoint2[24801] = {X 9.8592, Y 35.0049, Z -3.8333, A 0.000, B 0.000, C 0.000 }
gfCNCPoint2[24802] = {X 8.7492, Y 35.0957, Z -3.8333, A 0.000, B 0.000, C 0.000 }
gfCNCPoint2[24803] = {X 7.6565, Y 35.3113, Z -3.8333, A 0.000, B 0.000, C 0.000 }
gfCNCPoint2[24804] = {X 7.6482, Y 35.3823, Z -3.8333, A 0.000, B 0.000, C 0.000 }
gfCNCPoint2[24805] = {X 7.6519, Y 35.4537, Z -3.8333, A 0.000, B 0.000, C 0.000 }
gfCNCPoint2[24806] = {X 7.7647, Y 36.0463, Z -3.8333, A 0.000, B 0.000, C 0.000 }
gfCNCPoint2[24807] = {X 8.0674, Y 36.5680, Z -3.8333, A 0.000, B 0.000, C 0.000 }
gfCNCPoint2[24808] = {X 8.5259, Y 36.9600, Z -3.8333, A 0.000, B 0.000, C 0.000 }
gfCNCPoint2[24809] = {X 9.2839, Y 37.3409, Z -3.8333, A 0.000, B 0.000, C 0.000 }
gfCNCPoint2[24810] = {X 10.0891, Y 37.6076, Z -3.8333, A 0.000, B 0.000, C 0.000 }
gfCNCPoint2[24811] = {X 11.3662, Y 37.8456, Z -3.8333, A 0.000, B 0.000, C 0.000 }
gfCNCPoint2[24812] = {X 12.6631, Y 37.9217, Z -3.8333, A 0.000, B 0.000, C 0.000 }
gfCNCPoint2[24813] = {X 13.9594, Y 37.8349, Z -3.8333, A 0.000, B 0.000, C 0.000 }
gfCNCPoint2[24814] = {X 15.2345, Y 37.5863, Z -3.8333, A 0.000, B 0.000, C 0.000 }
gfCNCPoint2[24815] = {X 16.4685, Y 37.1800, Z -3.8333, A 0.000, B 0.000, C 0.000 }
gfCNCPoint2[24816] = {X 17.7887, Y 36.5661, Z -3.8333, A 0.000, B 0.000, C 0.000 }
gfCNCPoint2[24817] = {X 19.0345, Y 35.8123, Z -3.8333, A 0.000, B 0.000, C 0.000 }
gfCNCPoint2[24818] = {X 19.1547, Y 34.9706, Z -3.8333, A 0.000, B 0.000, C 0.000 }
gfCNCPoint2[24819] = {X 19.4346, Y 34.1678, Z -3.8333, A 0.000, B 0.000, C 0.000 }
gfCNCPoint2[24820] = {X 17.7798, Y 34.4462, Z -3.8333, A 0.000, B 0.000, C 0.000 }
gfCNCPoint2[24821] = {X 16.1107, Y 34.6192, Z -3.8333, A 0.000, B 0.000, C 0.000 }
gfCNCPoint2[24822] = {X 15.3859, Y 34.6719, Z -3.8333, A 0.000, B 0.000, C 0.000 }
gfCNCPoint2[24823] = {X 14.6610, Y 34.7226, Z -3.8333, A 0.000, B 0.000, C 0.000 }
gfCNCPoint2[24824] = {X 18.6548, Y 34.7187, Z -3.8333, A 0.000, B 0.000, C 0.000 }
gfCNCPoint2[24825] = {X 14.6555, Y 34.6427, Z -3.8333, A 0.000, B 0.000, C 0.000 }
gfCNCPoint2[24826] = {X 12.2590, Y 34.7952, Z -3.8333, A 0.000, B 0.000, C 0.000 }
gfCNCPoint2[24827] = {X 9.8611, Y 34.9248, Z -3.8333, A 0.000, B 0.000, C 0.000 }
gfCNCPoint2[24828] = {X 8.7163, Y 35.0195, Z -3.8333, A 0.000, B 0.000, C 0.000 }
gfCNCPoint2[24829] = {X 7.5902, Y 35.2458, Z -3.8333, A 0.000, B 0.000, C 0.000 }
gfCNCPoint2[24830] = {X 7.5711, Y 35.3439, Z -3.8333, A 0.000, B 0.000, C 0.000 }
gfCNCPoint2[24831] = {X 7.5717, Y 35.4438, Z -3.8333, A 0.000, B 0.000, C 0.000 }
gfCNCPoint2[24832] = {X 7.6871, Y 36.0671, Z -3.8333, A 0.000, B 0.000, C 0.000 }
gfCNCPoint2[24833] = {X 8.0035, Y 36.6163, Z -3.8333, A 0.000, B 0.000, C 0.000 }
gfCNCPoint2[24834] = {X 8.4849, Y 37.0287, Z -3.8333, A 0.000, B 0.000, C 0.000 }
gfCNCPoint2[24835] = {X 9.2532, Y 37.4148, Z -3.8333, A 0.000, B 0.000, C 0.000 }
gfCNCPoint2[24836] = {X 10.0695, Y 37.6852, Z -3.8333, A 0.000, B 0.000, C 0.000 }
gfCNCPoint2[24837] = {X 11.3565, Y 37.9250, Z -3.8333, A 0.000, B 0.000, C 0.000 }
gfCNCPoint2[24838] = {X 12.6634, Y 38.0017, Z -3.8333, A 0.000, B 0.000, C 0.000 }
gfCNCPoint2[24839] = {X 13.9697, Y 37.9142, Z -3.8333, A 0.000, B 0.000, C 0.000 }
gfCNCPoint2[24840] = {X 15.2547, Y 37.6637, Z -3.8333, A 0.000, B 0.000, C 0.000 }
gfCNCPoint2[24841] = {X 16.4982, Y 37.2543, Z -3.8333, A 0.000, B 0.000, C 0.000 }
gfCNCPoint2[24842] = {X 17.8441, Y 36.6272, Z -3.8333, A 0.000, B 0.000, C 0.000 }
gfCNCPoint2[24843] = {X 19.1128, Y 35.8557, Z -3.8333, A 0.000, B 0.000, C 0.000 }
gfCNCPoint2[24844] = {X 19.2471, Y 34.9311, Z -3.8333, A 0.000, B 0.000, C 0.000 }
gfCNCPoint2[24845] = {X 19.5771, Y 34.0571, Z -3.8333, A 0.000, B 0.000, C 0.000 }
gfCNCPoint2[24846] = {X 17.8490, Y 34.3560, Z -3.8333, A 0.000, B 0.000, C 0.000 }
gfCNCPoint2[24847] = {X 16.1049, Y 34.5394, Z -3.8333, A 0.000, B 0.000, C 0.000 }
gfCNCPoint2[24848] = {X 15.3803, Y 34.5921, Z -3.8333, A 0.000, B 0.000, C 0.000 }
gfCNCPoint2[24849] = {X 14.6555, Y 34.6427, Z -3.8333, A 0.000, B 0.000, C 0.000 }
gfCNCPoint2[24850] = {X 10.7038, Y 35.2624, Z -3.8333, A 0.000, B 0.000, C 0.000 }
gfCNCPoint2[24851] = {X 18.6493, Y 34.6389, Z -3.8333, A 0.000, B 0.000, C 0.000 }
gfCNCPoint2[24852] = {X 14.6501, Y 34.5629, Z -3.8333, A 0.000, B 0.000, C 0.000 }
gfCNCPoint2[24853] = {X 12.2548, Y 34.7153, Z -3.8333, A 0.000, B 0.000, C 0.000 }
gfCNCPoint2[24854] = {X 9.8581, Y 34.8448, Z -3.8333, A 0.000, B 0.000, C 0.000 }
gfCNCPoint2[24855] = {X 8.6835, Y 34.9434, Z -3.8333, A 0.000, B 0.000, C 0.000 }
gfCNCPoint2[24856] = {X 7.5285, Y 35.1794, Z -3.8333, A 0.000, B 0.000, C 0.000 }
gfCNCPoint2[24857] = {X 7.4943, Y 35.3117, Z -3.8333, A 0.000, B 0.000, C 0.000 }
gfCNCPoint2[24858] = {X 7.4918, Y 35.4484, Z -3.8333, A 0.000, B 0.000, C 0.000 }
gfCNCPoint2[24859] = {X 7.6128, Y 36.0970, Z -3.8333, A 0.000, B 0.000, C 0.000 }
gfCNCPoint2[24860] = {X 7.9427, Y 36.6683, Z -3.8333, A 0.000, B 0.000, C 0.000 }
gfCNCPoint2[24861] = {X 8.4439, Y 37.0974, Z -3.8333, A 0.000, B 0.000, C 0.000 }
gfCNCPoint2[24862] = {X 9.2226, Y 37.4887, Z -3.8333, A 0.000, B 0.000, C 0.000 }
gfCNCPoint2[24863] = {X 10.0499, Y 37.7628, Z -3.8333, A 0.000, B 0.000, C 0.000 }
gfCNCPoint2[24864] = {X 11.3468, Y 38.0044, Z -3.8333, A 0.000, B 0.000, C 0.000 }
gfCNCPoint2[24865] = {X 12.6638, Y 38.0817, Z -3.8333, A 0.000, B 0.000, C 0.000 }
gfCNCPoint2[24866] = {X 13.9800, Y 37.9935, Z -3.8333, A 0.000, B 0.000, C 0.000 }
gfCNCPoint2[24867] = {X 15.2749, Y 37.7411, Z -3.8333, A 0.000, B 0.000, C 0.000 }
gfCNCPoint2[24868] = {X 16.5279, Y 37.3285, Z -3.8333, A 0.000, B 0.000, C 0.000 }
gfCNCPoint2[24869] = {X 17.8997, Y 36.6881, Z -3.8333, A 0.000, B 0.000, C 0.000 }
gfCNCPoint2[24870] = {X 19.1915, Y 35.8986, Z -3.8333, A 0.000, B 0.000, C 0.000 }
gfCNCPoint2[24871] = {X 19.2643, Y 35.2208, Z -3.8333, A 0.000, B 0.000, C 0.000 }
gfCNCPoint2[24872] = {X 19.4447, Y 34.5634, Z -3.8333, A 0.000, B 0.000, C 0.000 }
gfCNCPoint2[24873] = {X 19.7282, Y 33.9435, Z -3.8333, A 0.000, B 0.000, C 0.000 }
gfCNCPoint2[24874] = {X 17.9226, Y 34.2648, Z -3.8333, A 0.000, B 0.000, C 0.000 }
gfCNCPoint2[24875] = {X 16.0990, Y 34.4596, Z -3.8333, A 0.000, B 0.000, C 0.000 }
gfCNCPoint2[24876] = {X 15.3746, Y 34.5123, Z -3.8333, A 0.000, B 0.000, C 0.000 }
gfCNCPoint2[24877] = {X 14.6501, Y 34.5629, Z -3.8333, A 0.000, B 0.000, C 0.000 }
gfCNCPoint2[24878] = {X 10.6983, Y 35.1826, Z -3.8333, A 0.000, B 0.000, C 0.000 }
gfCNCPoint2[24879] = {X 18.6439, Y 34.5591, Z -3.8333, A 0.000, B 0.000, C 0.000 }
gfCNCPoint2[24880] = {X 14.6446, Y 34.4831, Z -3.8333, A 0.000, B 0.000, C 0.000 }
gfCNCPoint2[24881] = {X 12.2505, Y 34.6354, Z -3.8333, A 0.000, B 0.000, C 0.000 }
gfCNCPoint2[24882] = {X 9.8552, Y 34.7649, Z -3.8333, A 0.000, B 0.000, C 0.000 }
gfCNCPoint2[24883] = {X 8.6523, Y 34.8670, Z -3.8333, A 0.000, B 0.000, C 0.000 }
gfCNCPoint2[24884] = {X 7.4702, Y 35.1122, Z -3.8333, A 0.000, B 0.000, C 0.000 }
gfCNCPoint2[24885] = {X 7.4185, Y 35.2786, Z -3.8333, A 0.000, B 0.000, C 0.000 }
gfCNCPoint2[24886] = {X 7.4119, Y 35.4528, Z -3.8333, A 0.000, B 0.000, C 0.000 }
gfCNCPoint2[24887] = {X 7.5385, Y 36.1267, Z -3.8333, A 0.000, B 0.000, C 0.000 }
gfCNCPoint2[24888] = {X 7.8818, Y 36.7203, Z -3.8333, A 0.000, B 0.000, C 0.000 }
gfCNCPoint2[24889] = {X 8.4028, Y 37.1661, Z -3.8333, A 0.000, B 0.000, C 0.000 }
gfCNCPoint2[24890] = {X 9.1920, Y 37.5626, Z -3.8333, A 0.000, B 0.000, C 0.000 }
gfCNCPoint2[24891] = {X 10.0304, Y 37.8403, Z -3.8333, A 0.000, B 0.000, C 0.000 }
gfCNCPoint2[24892] = {X 11.3371, Y 38.0838, Z -3.8333, A 0.000, B 0.000, C 0.000 }
gfCNCPoint2[24893] = {X 12.6641, Y 38.1617, Z -3.8333, A 0.000, B 0.000, C 0.000 }
gfCNCPoint2[24894] = {X 13.9904, Y 38.0728, Z -3.8333, A 0.000, B 0.000, C 0.000 }
gfCNCPoint2[24895] = {X 15.2951, Y 37.8185, Z -3.8333, A 0.000, B 0.000, C 0.000 }
gfCNCPoint2[24896] = {X 16.5577, Y 37.4028, Z -3.8333, A 0.000, B 0.000, C 0.000 }
gfCNCPoint2[24897] = {X 17.9556, Y 36.7489, Z -3.8333, A 0.000, B 0.000, C 0.000 }
gfCNCPoint2[24898] = {X 19.2706, Y 35.9411, Z -3.8333, A 0.000, B 0.000, C 0.000 }
gfCNCPoint2[24899] = {X 19.3492, Y 35.2029, Z -3.8333, A 0.000, B 0.000, C 0.000 }
gfCNCPoint2[24900] = {X 19.5578, Y 34.4904, Z -3.8333, A 0.000, B 0.000, C 0.000 }
gfCNCPoint2[24901] = {X 19.8898, Y 33.8264, Z -3.8333, A 0.000, B 0.000, C 0.000 }
gfCNCPoint2[24902] = {X 18.0016, Y 34.1726, Z -3.8333, A 0.000, B 0.000, C 0.000 }
gfCNCPoint2[24903] = {X 16.0932, Y 34.3799, Z -3.8333, A 0.000, B 0.000, C 0.000 }
gfCNCPoint2[24904] = {X 15.3690, Y 34.4325, Z -3.8333, A 0.000, B 0.000, C 0.000 }
gfCNCPoint2[24905] = {X 14.6446, Y 34.4831, Z -3.8333, A 0.000, B 0.000, C 0.000 }
gfCNCPoint2[24906] = {X 10.6929, Y 35.1028, Z -3.8333, A 0.000, B 0.000, C 0.000 }
gfCNCPoint2[24907] = {X 18.6384, Y 34.4793, Z -3.8333, A 0.000, B 0.000, C 0.000 }
gfCNCPoint2[24908] = {X 14.6391, Y 34.4033, Z -3.8333, A 0.000, B 0.000, C 0.000 }
gfCNCPoint2[24909] = {X 12.2463, Y 34.5555, Z -3.8333, A 0.000, B 0.000, C 0.000 }
gfCNCPoint2[24910] = {X 9.8522, Y 34.6849, Z -3.8333, A 0.000, B 0.000, C 0.000 }
gfCNCPoint2[24911] = {X 8.6224, Y 34.7906, Z -3.8333, A 0.000, B 0.000, C 0.000 }
gfCNCPoint2[24912] = {X 7.4145, Y 35.0445, Z -3.8333, A 0.000, B 0.000, C 0.000 }
gfCNCPoint2[24913] = {X 7.3434, Y 35.2448, Z -3.8333, A 0.000, B 0.000, C 0.000 }
gfCNCPoint2[24914] = {X 7.3319, Y 35.4571, Z -3.8333, A 0.000, B 0.000, C 0.000 }
gfCNCPoint2[24915] = {X 7.4091, Y 35.9864, Z -3.8333, A 0.000, B 0.000, C 0.000 }
gfCNCPoint2[24916] = {X 7.6165, Y 36.4794, Z -3.8333, A 0.000, B 0.000, C 0.000 }
gfCNCPoint2[24917] = {X 7.9410, Y 36.9046, Z -3.8333, A 0.000, B 0.000, C 0.000 }
gfCNCPoint2[24918] = {X 8.3618, Y 37.2348, Z -3.8333, A 0.000, B 0.000, C 0.000 }
gfCNCPoint2[24919] = {X 9.1614, Y 37.6365, Z -3.8333, A 0.000, B 0.000, C 0.000 }
gfCNCPoint2[24920] = {X 10.0108, Y 37.9179, Z -3.8333, A 0.000, B 0.000, C 0.000 }
gfCNCPoint2[24921] = {X 11.3275, Y 38.1632, Z -3.8333, A 0.000, B 0.000, C 0.000 }
gfCNCPoint2[24922] = {X 12.6644, Y 38.2417, Z -3.8333, A 0.000, B 0.000, C 0.000 }
gfCNCPoint2[24923] = {X 14.0007, Y 38.1522, Z -3.8333, A 0.000, B 0.000, C 0.000 }
gfCNCPoint2[24924] = {X 15.3153, Y 37.8959, Z -3.8333, A 0.000, B 0.000, C 0.000 }
gfCNCPoint2[24925] = {X 16.5874, Y 37.4771, Z -3.8333, A 0.000, B 0.000, C 0.000 }
gfCNCPoint2[24926] = {X 18.0117, Y 36.8095, Z -3.8333, A 0.000, B 0.000, C 0.000 }
gfCNCPoint2[24927] = {X 19.3501, Y 35.9832, Z -3.8333, A 0.000, B 0.000, C 0.000 }
gfCNCPoint2[24928] = {X 19.4352, Y 35.1814, Z -3.8333, A 0.000, B 0.000, C 0.000 }
gfCNCPoint2[24929] = {X 19.6763, Y 34.4120, Z -3.8333, A 0.000, B 0.000, C 0.000 }
gfCNCPoint2[24930] = {X 20.0641, Y 33.7051, Z -3.8333, A 0.000, B 0.000, C 0.000 }
gfCNCPoint2[24931] = {X 18.0872, Y 34.0791, Z -3.8333, A 0.000, B 0.000, C 0.000 }
gfCNCPoint2[24932] = {X 16.0874, Y 34.3001, Z -3.8333, A 0.000, B 0.000, C 0.000 }
gfCNCPoint2[24933] = {X 15.3633, Y 34.3527, Z -3.8333, A 0.000, B 0.000, C 0.000 }
gfCNCPoint2[24934] = {X 14.6391, Y 34.4033, Z -3.8333, A 0.000, B 0.000, C 0.000 }
gfCNCPoint2[24935] = {X 10.6874, Y 35.0230, Z -3.8333, A 0.000, B 0.000, C 0.000 }
gfCNCPoint2[24936] = {X 14.7701, Y 36.3188, Z -3.8333, A 0.000, B 0.000, C 0.000 }
gfCNCPoint2[24937] = {X 14.6337, Y 34.3235, Z -3.8333, A 0.000, B 0.000, C 0.000 }
gfCNCPoint2[24938] = {X 12.2421, Y 34.4756, Z -3.8333, A 0.000, B 0.000, C 0.000 }
gfCNCPoint2[24939] = {X 9.8492, Y 34.6050, Z -3.8333, A 0.000, B 0.000, C 0.000 }
gfCNCPoint2[24940] = {X 8.5936, Y 34.7140, Z -3.8333, A 0.000, B 0.000, C 0.000 }
gfCNCPoint2[24941] = {X 7.3608, Y 34.9763, Z -3.8333, A 0.000, B 0.000, C 0.000 }
gfCNCPoint2[24942] = {X 7.2689, Y 35.2104, Z -3.8333, A 0.000, B 0.000, C 0.000 }
gfCNCPoint2[24943] = {X 7.2520, Y 35.4613, Z -3.8333, A 0.000, B 0.000, C 0.000 }
gfCNCPoint2[24944] = {X 7.3325, Y 36.0099, Z -3.8333, A 0.000, B 0.000, C 0.000 }
gfCNCPoint2[24945] = {X 7.5480, Y 36.5207, Z -3.8333, A 0.000, B 0.000, C 0.000 }
gfCNCPoint2[24946] = {X 7.8846, Y 36.9613, Z -3.8333, A 0.000, B 0.000, C 0.000 }
gfCNCPoint2[24947] = {X 8.3208, Y 37.3034, Z -3.8333, A 0.000, B 0.000, C 0.000 }
gfCNCPoint2[24948] = {X 9.1308, Y 37.7104, Z -3.8333, A 0.000, B 0.000, C 0.000 }
gfCNCPoint2[24949] = {X 9.9913, Y 37.9955, Z -3.8333, A 0.000, B 0.000, C 0.000 }
gfCNCPoint2[24950] = {X 11.3178, Y 38.2426, Z -3.8333, A 0.000, B 0.000, C 0.000 }
gfCNCPoint2[24951] = {X 12.6648, Y 38.3217, Z -3.8333, A 0.000, B 0.000, C 0.000 }
gfCNCPoint2[24952] = {X 14.0111, Y 38.2315, Z -3.8333, A 0.000, B 0.000, C 0.000 }
gfCNCPoint2[24953] = {X 15.3355, Y 37.9733, Z -3.8333, A 0.000, B 0.000, C 0.000 }
gfCNCPoint2[24954] = {X 16.6172, Y 37.5514, Z -3.8333, A 0.000, B 0.000, C 0.000 }
gfCNCPoint2[24955] = {X 18.0680, Y 36.8700, Z -3.8333, A 0.000, B 0.000, C 0.000 }
gfCNCPoint2[24956] = {X 19.4300, Y 36.0248, Z -3.8333, A 0.000, B 0.000, C 0.000 }
gfCNCPoint2[24957] = {X 19.5226, Y 35.1553, Z -3.8333, A 0.000, B 0.000, C 0.000 }
gfCNCPoint2[24958] = {X 19.8019, Y 34.3266, Z -3.8333, A 0.000, B 0.000, C 0.000 }
gfCNCPoint2[24959] = {X 20.2547, Y 33.5784, Z -3.8333, A 0.000, B 0.000, C 0.000 }
gfCNCPoint2[24960] = {X 18.1811, Y 33.9840, Z -3.8333, A 0.000, B 0.000, C 0.000 }
gfCNCPoint2[24961] = {X 16.0816, Y 34.2203, Z -3.8333, A 0.000, B 0.000, C 0.000 }
gfCNCPoint2[24962] = {X 15.3577, Y 34.2729, Z -3.8333, A 0.000, B 0.000, C 0.000 }
gfCNCPoint2[24963] = {X 14.6337, Y 34.3235, Z -3.8333, A 0.000, B 0.000, C 0.000 }
gfCNCPoint2[24964] = {X 14.7701, Y 36.3188, Z -3.8333, A 0.000, B 0.000, C 0.000 }
gfCNCPoint2[24965] = {X 14.7701, Y 36.3188, Z -0.8333, A 0.000, B 0.000, C 0.000 }
gfCNCPoint2[24966] = {X 14.7701, Y 36.3188, Z 11.0000, A 0.000, B 0.000, C 0.000 }
gfCNCPoint2[24967] = {X 165.6772, Y 73.8165, Z 11.0000, A 0.000, B 0.000, C 0.000 }
gfCNCPoint2[24968] = {X 165.6772, Y 73.8165, Z 0.0000, A 0.000, B 0.000, C 0.000 }
gfCNCPoint2[24969] = {X 161.3996, Y 78.5670, Z -1.7129, A 0.000, B 0.000, C 0.000 }
gfCNCPoint2[24970] = {X 169.3132, Y 78.5670, Z -3.8333, A 0.000, B 0.000, C 0.000 }
gfCNCPoint2[24971] = {X 169.3132, Y 76.1670, Z -3.8333, A 0.000, B 0.000, C 0.000 }
gfCNCPoint2[24972] = {X 171.8361, Y 76.1670, Z -3.8333, A 0.000, B 0.000, C 0.000 }
gfCNCPoint2[24973] = {X 169.3147, Y 73.3634, Z -3.8333, A 0.000, B 0.000, C 0.000 }
gfCNCPoint2[24974] = {X 166.7903, Y 76.1670, Z -3.8333, A 0.000, B 0.000, C 0.000 }
gfCNCPoint2[24975] = {X 169.3132, Y 76.1670, Z -3.8333, A 0.000, B 0.000, C 0.000 }
gfCNCPoint2[24976] = {X 169.3132, Y 78.5670, Z -3.8333, A 0.000, B 0.000, C 0.000 }
gfCNCPoint2[24977] = {X 177.2224, Y 78.5670, Z -3.8333, A 0.000, B 0.000, C 0.000 }
gfCNCPoint2[24978] = {X 169.3158, Y 69.7756, Z -3.8333, A 0.000, B 0.000, C 0.000 }
gfCNCPoint2[24979] = {X 161.3996, Y 78.5670, Z -3.8333, A 0.000, B 0.000, C 0.000 }
gfCNCPoint2[24980] = {X 169.3132, Y 78.5670, Z -3.8333, A 0.000, B 0.000, C 0.000 }
gfCNCPoint2[24981] = {X 169.3132, Y 74.6470, Z -3.8333, A 0.000, B 0.000, C 0.000 }
gfCNCPoint2[24982] = {X 169.3132, Y 78.6470, Z -3.8333, A 0.000, B 0.000, C 0.000 }
gfCNCPoint2[24983] = {X 177.4019, Y 78.6470, Z -3.8333, A 0.000, B 0.000, C 0.000 }
gfCNCPoint2[24984] = {X 169.3159, Y 69.6560, Z -3.8333, A 0.000, B 0.000, C 0.000 }
gfCNCPoint2[24985] = {X 161.2199, Y 78.6470, Z -3.8333, A 0.000, B 0.000, C 0.000 }
gfCNCPoint2[24986] = {X 169.3132, Y 78.6470, Z -3.8333, A 0.000, B 0.000, C 0.000 }
gfCNCPoint2[24987] = {X 169.3132, Y 74.6470, Z -3.8333, A 0.000, B 0.000, C 0.000 }
gfCNCPoint2[24988] = {X 169.3132, Y 74.7270, Z -3.8333, A 0.000, B 0.000, C 0.000 }
gfCNCPoint2[24989] = {X 169.3132, Y 78.7270, Z -3.8333, A 0.000, B 0.000, C 0.000 }
gfCNCPoint2[24990] = {X 177.5814, Y 78.7270, Z -3.8333, A 0.000, B 0.000, C 0.000 }
gfCNCPoint2[24991] = {X 169.3159, Y 69.5364, Z -3.8333, A 0.000, B 0.000, C 0.000 }
gfCNCPoint2[24992] = {X 161.0403, Y 78.7270, Z -3.8333, A 0.000, B 0.000, C 0.000 }
gfCNCPoint2[24993] = {X 169.3132, Y 78.7270, Z -3.8333, A 0.000, B 0.000, C 0.000 }
gfCNCPoint2[24994] = {X 169.3132, Y 74.7270, Z -3.8333, A 0.000, B 0.000, C 0.000 }
gfCNCPoint2[24995] = {X 169.3132, Y 74.8070, Z -3.8333, A 0.000, B 0.000, C 0.000 }
gfCNCPoint2[24996] = {X 169.3132, Y 78.8070, Z -3.8333, A 0.000, B 0.000, C 0.000 }
gfCNCPoint2[24997] = {X 177.7610, Y 78.8070, Z -3.8333, A 0.000, B 0.000, C 0.000 }
gfCNCPoint2[24998] = {X 169.3159, Y 69.4168, Z -3.8333, A 0.000, B 0.000, C 0.000 }
gfCNCPoint2[24999] = {X 160.8606, Y 78.8070, Z -3.8333, A 0.000, B 0.000, C 0.000 }
gfCNCPoint2[25000] = {X 169.3132, Y 78.8070, Z -3.8333, A 0.000, B 0.000, C 0.000 }
gfCNCPoint2[25001] = {X 169.3132, Y 74.8070, Z -3.8333, A 0.000, B 0.000, C 0.000 }
gfCNCPoint2[25002] = {X 169.3132, Y 74.8870, Z -3.8333, A 0.000, B 0.000, C 0.000 }
gfCNCPoint2[25003] = {X 169.3132, Y 78.8870, Z -3.8333, A 0.000, B 0.000, C 0.000 }
gfCNCPoint2[25004] = {X 177.9405, Y 78.8870, Z -3.8333, A 0.000, B 0.000, C 0.000 }
gfCNCPoint2[25005] = {X 169.3160, Y 69.2972, Z -3.8333, A 0.000, B 0.000, C 0.000 }
gfCNCPoint2[25006] = {X 160.6809, Y 78.8870, Z -3.8333, A 0.000, B 0.000, C 0.000 }
gfCNCPoint2[25007] = {X 169.3132, Y 78.8870, Z -3.8333, A 0.000, B 0.000, C 0.000 }
gfCNCPoint2[25008] = {X 169.3132, Y 74.8870, Z -3.8333, A 0.000, B 0.000, C 0.000 }
gfCNCPoint2[25009] = {X 169.3132, Y 74.9670, Z -3.8333, A 0.000, B 0.000, C 0.000 }
gfCNCPoint2[25010] = {X 169.3132, Y 78.9670, Z -3.8333, A 0.000, B 0.000, C 0.000 }
gfCNCPoint2[25011] = {X 178.1201, Y 78.9670, Z -3.8333, A 0.000, B 0.000, C 0.000 }
gfCNCPoint2[25012] = {X 169.3160, Y 69.1776, Z -3.8333, A 0.000, B 0.000, C 0.000 }
gfCNCPoint2[25013] = {X 160.5012, Y 78.9670, Z -3.8333, A 0.000, B 0.000, C 0.000 }
gfCNCPoint2[25014] = {X 169.3132, Y 78.9670, Z -3.8333, A 0.000, B 0.000, C 0.000 }
gfCNCPoint2[25015] = {X 169.3132, Y 74.9670, Z -3.8333, A 0.000, B 0.000, C 0.000 }
gfCNCPoint2[25016] = {X 169.3132, Y 74.9670, Z -0.8333, A 0.000, B 0.000, C 0.000 }
gfCNCPoint2[25017] = {X 169.3132, Y 74.9670, Z 11.0000, A 0.000, B 0.000, C 0.000 }
gfCNCPoint2[25018] = {X 186.2298, Y 37.9125, Z 11.0000, A 0.000, B 0.000, C 0.000 }
gfCNCPoint2[25019] = {X 186.2298, Y 37.9125, Z 0.0000, A 0.000, B 0.000, C 0.000 }
gfCNCPoint2[25020] = {X 187.5911, Y 37.8326, Z -0.3654, A 0.000, B 0.000, C 0.000 }
gfCNCPoint2[25021] = {X 189.4187, Y 37.3859, Z -0.8695, A 0.000, B 0.000, C 0.000 }
gfCNCPoint2[25022] = {X 190.1439, Y 37.0739, Z -1.0811, A 0.000, B 0.000, C 0.000 }
gfCNCPoint2[25023] = {X 190.9812, Y 36.7137, Z -1.3253, A 0.000, B 0.000, C 0.000 }
gfCNCPoint2[25024] = {X 191.6925, Y 36.3239, Z -1.5426, A 0.000, B 0.000, C 0.000 }
gfCNCPoint2[25025] = {X 192.4466, Y 35.8119, Z -1.7869, A 0.000, B 0.000, C 0.000 }
gfCNCPoint2[25026] = {X 192.4699, Y 35.2977, Z -1.9248, A 0.000, B 0.000, C 0.000 }
gfCNCPoint2[25027] = {X 192.6315, Y 34.6343, Z -2.1077, A 0.000, B 0.000, C 0.000 }
gfCNCPoint2[25028] = {X 192.8472, Y 34.1670, Z -2.2457, A 0.000, B 0.000, C 0.000 }
gfCNCPoint2[25029] = {X 192.7390, Y 34.1922, Z -2.2754, A 0.000, B 0.000, C 0.000 }
gfCNCPoint2[25030] = {X 191.4095, Y 34.4424, Z -2.6379, A 0.000, B 0.000, C 0.000 }
gfCNCPoint2[25031] = {X 190.5800, Y 34.5491, Z -2.8620, A 0.000, B 0.000, C 0.000 }
gfCNCPoint2[25032] = {X 189.2271, Y 34.6439, Z -3.2254, A 0.000, B 0.000, C 0.000 }
gfCNCPoint2[25033] = {X 186.9626, Y 34.7829, Z -3.8333, A 0.000, B 0.000, C 0.000 }
gfCNCPoint2[25034] = {X 182.5757, Y 35.0523, Z -3.8333, A 0.000, B 0.000, C 0.000 }
gfCNCPoint2[25035] = {X 181.8173, Y 35.1397, Z -3.8333, A 0.000, B 0.000, C 0.000 }
gfCNCPoint2[25036] = {X 181.0726, Y 35.3077, Z -3.8333, A 0.000, B 0.000, C 0.000 }
gfCNCPoint2[25037] = {X 181.0644, Y 35.3821, Z -3.8333, A 0.000, B 0.000, C 0.000 }
gfCNCPoint2[25038] = {X 181.0644, Y 35.4568, Z -3.8333, A 0.000, B 0.000, C 0.000 }
gfCNCPoint2[25039] = {X 181.1573, Y 36.0000, Z -3.8333, A 0.000, B 0.000, C 0.000 }
gfCNCPoint2[25040] = {X 181.4146, Y 36.4873, Z -3.8333, A 0.000, B 0.000, C 0.000 }
gfCNCPoint2[25041] = {X 181.8107, Y 36.8704, Z -3.8333, A 0.000, B 0.000, C 0.000 }
gfCNCPoint2[25042] = {X 182.4284, Y 37.2231, Z -3.8333, A 0.000, B 0.000, C 0.000 }
gfCNCPoint2[25043] = {X 183.0887, Y 37.4879, Z -3.8333, A 0.000, B 0.000, C 0.000 }
gfCNCPoint2[25044] = {X 184.4953, Y 37.8017, Z -3.8333, A 0.000, B 0.000, C 0.000 }
gfCNCPoint2[25045] = {X 185.9318, Y 37.9176, Z -3.8333, A 0.000, B 0.000, C 0.000 }
gfCNCPoint2[25046] = {X 187.3705, Y 37.8331, Z -3.8333, A 0.000, B 0.000, C 0.000 }
gfCNCPoint2[25047] = {X 188.7837, Y 37.5501, Z -3.8333, A 0.000, B 0.000, C 0.000 }
gfCNCPoint2[25048] = {X 190.1439, Y 37.0739, Z -3.8333, A 0.000, B 0.000, C 0.000 }
gfCNCPoint2[25049] = {X 191.3253, Y 36.4977, Z -3.8333, A 0.000, B 0.000, C 0.000 }
gfCNCPoint2[25050] = {X 192.4466, Y 35.8119, Z -3.8333, A 0.000, B 0.000, C 0.000 }
gfCNCPoint2[25051] = {X 192.5671, Y 34.9700, Z -3.8333, A 0.000, B 0.000, C 0.000 }
gfCNCPoint2[25052] = {X 192.8472, Y 34.1670, Z -3.8333, A 0.000, B 0.000, C 0.000 }
gfCNCPoint2[25053] = {X 192.7390, Y 34.1922, Z -3.8333, A 0.000, B 0.000, C 0.000 }
gfCNCPoint2[25054] = {X 190.9896, Y 34.4691, Z -3.8333, A 0.000, B 0.000, C 0.000 }
gfCNCPoint2[25055] = {X 189.2271, Y 34.6439, Z -3.8333, A 0.000, B 0.000, C 0.000 }
gfCNCPoint2[25056] = {X 186.9626, Y 34.7829, Z -3.8333, A 0.000, B 0.000, C 0.000 }
gfCNCPoint2[25057] = {X 190.9563, Y 34.8068, Z -3.8333, A 0.000, B 0.000, C 0.000 }
gfCNCPoint2[25058] = {X 186.9577, Y 34.7031, Z -3.8333, A 0.000, B 0.000, C 0.000 }
gfCNCPoint2[25059] = {X 182.5708, Y 34.9724, Z -3.8333, A 0.000, B 0.000, C 0.000 }
gfCNCPoint2[25060] = {X 181.7797, Y 35.0650, Z -3.8333, A 0.000, B 0.000, C 0.000 }
gfCNCPoint2[25061] = {X 181.0036, Y 35.2442, Z -3.8333, A 0.000, B 0.000, C 0.000 }
gfCNCPoint2[25062] = {X 180.9868, Y 35.3480, Z -3.8333, A 0.000, B 0.000, C 0.000 }
gfCNCPoint2[25063] = {X 180.9844, Y 35.4530, Z -3.8333, A 0.000, B 0.000, C 0.000 }
gfCNCPoint2[25064] = {X 181.0807, Y 36.0230, Z -3.8333, A 0.000, B 0.000, C 0.000 }
gfCNCPoint2[25065] = {X 181.3500, Y 36.5346, Z -3.8333, A 0.000, B 0.000, C 0.000 }
gfCNCPoint2[25066] = {X 181.7656, Y 36.9365, Z -3.8333, A 0.000, B 0.000, C 0.000 }
gfCNCPoint2[25067] = {X 182.3936, Y 37.2952, Z -3.8333, A 0.000, B 0.000, C 0.000 }
gfCNCPoint2[25068] = {X 183.0650, Y 37.5643, Z -3.8333, A 0.000, B 0.000, C 0.000 }
gfCNCPoint2[25069] = {X 184.4826, Y 37.8807, Z -3.8333, A 0.000, B 0.000, C 0.000 }
gfCNCPoint2[25070] = {X 185.9304, Y 37.9975, Z -3.8333, A 0.000, B 0.000, C 0.000 }
gfCNCPoint2[25071] = {X 187.3804, Y 37.9125, Z -3.8333, A 0.000, B 0.000, C 0.000 }
gfCNCPoint2[25072] = {X 188.8046, Y 37.6273, Z -3.8333, A 0.000, B 0.000, C 0.000 }
gfCNCPoint2[25073] = {X 190.1755, Y 37.1474, Z -3.8333, A 0.000, B 0.000, C 0.000 }
gfCNCPoint2[25074] = {X 191.3814, Y 36.5581, Z -3.8333, A 0.000, B 0.000, C 0.000 }
gfCNCPoint2[25075] = {X 192.5249, Y 35.8554, Z -3.8333, A 0.000, B 0.000, C 0.000 }
gfCNCPoint2[25076] = {X 192.6603, Y 34.9273, Z -3.8333, A 0.000, B 0.000, C 0.000 }
gfCNCPoint2[25077] = {X 192.9927, Y 34.0502, Z -3.8333, A 0.000, B 0.000, C 0.000 }
gfCNCPoint2[25078] = {X 192.7315, Y 34.1122, Z -3.8333, A 0.000, B 0.000, C 0.000 }
gfCNCPoint2[25079] = {X 190.9841, Y 34.3891, Z -3.8333, A 0.000, B 0.000, C 0.000 }
gfCNCPoint2[25080] = {X 189.2235, Y 34.5639, Z -3.8333, A 0.000, B 0.000, C 0.000 }
gfCNCPoint2[25081] = {X 186.9577, Y 34.7031, Z -3.8333, A 0.000, B 0.000, C 0.000 }
gfCNCPoint2[25082] = {X 183.0017, Y 35.2952, Z -3.8333, A 0.000, B 0.000, C 0.000 }
gfCNCPoint2[25083] = {X 190.9514, Y 34.7270, Z -3.8333, A 0.000, B 0.000, C 0.000 }
gfCNCPoint2[25084] = {X 186.9528, Y 34.6232, Z -3.8333, A 0.000, B 0.000, C 0.000 }
gfCNCPoint2[25085] = {X 182.5659, Y 34.8926, Z -3.8333, A 0.000, B 0.000, C 0.000 }
gfCNCPoint2[25086] = {X 181.7437, Y 34.9901, Z -3.8333, A 0.000, B 0.000, C 0.000 }
gfCNCPoint2[25087] = {X 180.9378, Y 35.1802, Z -3.8333, A 0.000, B 0.000, C 0.000 }
gfCNCPoint2[25088] = {X 180.9098, Y 35.3163, Z -3.8333, A 0.000, B 0.000, C 0.000 }
gfCNCPoint2[25089] = {X 180.9044, Y 35.4551, Z -3.8333, A 0.000, B 0.000, C 0.000 }
gfCNCPoint2[25090] = {X 181.0053, Y 36.0498, Z -3.8333, A 0.000, B 0.000, C 0.000 }
gfCNCPoint2[25091] = {X 181.2867, Y 36.5834, Z -3.8333, A 0.000, B 0.000, C 0.000 }
gfCNCPoint2[25092] = {X 181.7205, Y 37.0025, Z -3.8333, A 0.000, B 0.000, C 0.000 }
gfCNCPoint2[25093] = {X 182.3589, Y 37.3672, Z -3.8333, A 0.000, B 0.000, C 0.000 }
gfCNCPoint2[25094] = {X 183.0413, Y 37.6407, Z -3.8333, A 0.000, B 0.000, C 0.000 }
gfCNCPoint2[25095] = {X 184.4699, Y 37.9597, Z -3.8333, A 0.000, B 0.000, C 0.000 }
gfCNCPoint2[25096] = {X 185.9290, Y 38.0775, Z -3.8333, A 0.000, B 0.000, C 0.000 }
gfCNCPoint2[25097] = {X 187.3903, Y 37.9919, Z -3.8333, A 0.000, B 0.000, C 0.000 }
gfCNCPoint2[25098] = {X 188.8256, Y 37.7045, Z -3.8333, A 0.000, B 0.000, C 0.000 }
gfCNCPoint2[25099] = {X 190.2072, Y 37.2209, Z -3.8333, A 0.000, B 0.000, C 0.000 }
gfCNCPoint2[25100] = {X 191.4378, Y 36.6184, Z -3.8333, A 0.000, B 0.000, C 0.000 }
gfCNCPoint2[25101] = {X 192.6036, Y 35.8984, Z -3.8333, A 0.000, B 0.000, C 0.000 }
gfCNCPoint2[25102] = {X 192.6773, Y 35.2162, Z -3.8333, A 0.000, B 0.000, C 0.000 }
gfCNCPoint2[25103] = {X 192.8601, Y 34.5547, Z -3.8333, A 0.000, B 0.000, C 0.000 }
gfCNCPoint2[25104] = {X 193.1471, Y 33.9314, Z -3.8333, A 0.000, B 0.000, C 0.000 }
gfCNCPoint2[25105] = {X 192.7149, Y 34.0339, Z -3.8333, A 0.000, B 0.000, C 0.000 }
gfCNCPoint2[25106] = {X 190.9731, Y 34.3099, Z -3.8333, A 0.000, B 0.000, C 0.000 }
gfCNCPoint2[25107] = {X 189.2183, Y 34.4841, Z -3.8333, A 0.000, B 0.000, C 0.000 }
gfCNCPoint2[25108] = {X 186.9528, Y 34.6232, Z -3.8333, A 0.000, B 0.000, C 0.000 }
gfCNCPoint2[25109] = {X 182.9968, Y 35.2154, Z -3.8333, A 0.000, B 0.000, C 0.000 }
gfCNCPoint2[25110] = {X 190.9465, Y 34.6471, Z -3.8333, A 0.000, B 0.000, C 0.000 }
gfCNCPoint2[25111] = {X 186.9479, Y 34.5434, Z -3.8333, A 0.000, B 0.000, C 0.000 }
gfCNCPoint2[25112] = {X 182.5610, Y 34.8127, Z -3.8333, A 0.000, B 0.000, C 0.000 }
gfCNCPoint2[25113] = {X 181.7089, Y 34.9150, Z -3.8333, A 0.000, B 0.000, C 0.000 }
gfCNCPoint2[25114] = {X 180.8745, Y 35.1156, Z -3.8333, A 0.000, B 0.000, C 0.000 }
gfCNCPoint2[25115] = {X 180.8334, Y 35.2841, Z -3.8333, A 0.000, B 0.000, C 0.000 }
gfCNCPoint2[25116] = {X 180.8244, Y 35.4572, Z -3.8333, A 0.000, B 0.000, C 0.000 }
gfCNCPoint2[25117] = {X 180.9299, Y 36.0766, Z -3.8333, A 0.000, B 0.000, C 0.000 }
gfCNCPoint2[25118] = {X 181.2233, Y 36.6323, Z -3.8333, A 0.000, B 0.000, C 0.000 }
gfCNCPoint2[25119] = {X 181.6754, Y 37.0686, Z -3.8333, A 0.000, B 0.000, C 0.000 }
gfCNCPoint2[25120] = {X 182.3241, Y 37.4393, Z -3.8333, A 0.000, B 0.000, C 0.000 }
gfCNCPoint2[25121] = {X 183.0176, Y 37.7171, Z -3.8333, A 0.000, B 0.000, C 0.000 }
gfCNCPoint2[25122] = {X 184.4572, Y 38.0387, Z -3.8333, A 0.000, B 0.000, C 0.000 }
gfCNCPoint2[25123] = {X 185.9275, Y 38.1575, Z -3.8333, A 0.000, B 0.000, C 0.000 }
gfCNCPoint2[25124] = {X 187.4001, Y 38.0713, Z -3.8333, A 0.000, B 0.000, C 0.000 }
gfCNCPoint2[25125] = {X 188.8465, Y 37.7817, Z -3.8333, A 0.000, B 0.000, C 0.000 }
gfCNCPoint2[25126] = {X 190.2388, Y 37.2944, Z -3.8333, A 0.000, B 0.000, C 0.000 }
gfCNCPoint2[25127] = {X 191.4944, Y 36.6785, Z -3.8333, A 0.000, B 0.000, C 0.000 }
gfCNCPoint2[25128] = {X 192.6827, Y 35.9411, Z -3.8333, A 0.000, B 0.000, C 0.000 }
gfCNCPoint2[25129] = {X 192.7626, Y 35.1966, Z -3.8333, A 0.000, B 0.000, C 0.000 }
gfCNCPoint2[25130] = {X 192.9747, Y 34.4785, Z -3.8333, A 0.000, B 0.000, C 0.000 }
gfCNCPoint2[25131] = {X 193.3120, Y 33.8101, Z -3.8333, A 0.000, B 0.000, C 0.000 }
gfCNCPoint2[25132] = {X 192.6983, Y 33.9556, Z -3.8333, A 0.000, B 0.000, C 0.000 }
gfCNCPoint2[25133] = {X 190.9622, Y 34.2306, Z -3.8333, A 0.000, B 0.000, C 0.000 }
gfCNCPoint2[25134] = {X 189.2131, Y 34.4043, Z -3.8333, A 0.000, B 0.000, C 0.000 }
gfCNCPoint2[25135] = {X 186.9479, Y 34.5434, Z -3.8333, A 0.000, B 0.000, C 0.000 }
gfCNCPoint2[25136] = {X 182.9919, Y 35.1355, Z -3.8333, A 0.000, B 0.000, C 0.000 }
gfCNCPoint2[25137] = {X 190.9416, Y 34.5673, Z -3.8333, A 0.000, B 0.000, C 0.000 }
gfCNCPoint2[25138] = {X 186.9429, Y 34.4635, Z -3.8333, A 0.000, B 0.000, C 0.000 }
gfCNCPoint2[25139] = {X 182.5561, Y 34.7329, Z -3.8333, A 0.000, B 0.000, C 0.000 }
gfCNCPoint2[25140] = {X 181.6752, Y 34.8399, Z -3.8333, A 0.000, B 0.000, C 0.000 }
gfCNCPoint2[25141] = {X 180.8132, Y 35.0507, Z -3.8333, A 0.000, B 0.000, C 0.000 }
gfCNCPoint2[25142] = {X 180.7575, Y 35.2514, Z -3.8333, A 0.000, B 0.000, C 0.000 }
gfCNCPoint2[25143] = {X 180.7444, Y 35.4593, Z -3.8333, A 0.000, B 0.000, C 0.000 }
gfCNCPoint2[25144] = {X 180.8545, Y 36.1034, Z -3.8333, A 0.000, B 0.000, C 0.000 }
gfCNCPoint2[25145] = {X 181.1600, Y 36.6811, Z -3.8333, A 0.000, B 0.000, C 0.000 }
gfCNCPoint2[25146] = {X 181.6303, Y 37.1347, Z -3.8333, A 0.000, B 0.000, C 0.000 }
gfCNCPoint2[25147] = {X 182.2893, Y 37.5113, Z -3.8333, A 0.000, B 0.000, C 0.000 }
gfCNCPoint2[25148] = {X 182.9939, Y 37.7936, Z -3.8333, A 0.000, B 0.000, C 0.000 }
gfCNCPoint2[25149] = {X 184.4445, Y 38.1177, Z -3.8333, A 0.000, B 0.000, C 0.000 }
gfCNCPoint2[25150] = {X 185.9261, Y 38.2375, Z -3.8333, A 0.000, B 0.000, C 0.000 }
gfCNCPoint2[25151] = {X 187.4100, Y 38.1507, Z -3.8333, A 0.000, B 0.000, C 0.000 }
gfCNCPoint2[25152] = {X 188.8674, Y 37.8589, Z -3.8333, A 0.000, B 0.000, C 0.000 }
gfCNCPoint2[25153] = {X 190.2704, Y 37.3679, Z -3.8333, A 0.000, B 0.000, C 0.000 }
gfCNCPoint2[25154] = {X 191.5513, Y 36.7385, Z -3.8333, A 0.000, B 0.000, C 0.000 }
gfCNCPoint2[25155] = {X 192.7622, Y 35.9833, Z -3.8333, A 0.000, B 0.000, C 0.000 }
gfCNCPoint2[25156] = {X 192.8358, Y 35.2390, Z -3.8333, A 0.000, B 0.000, C 0.000 }
gfCNCPoint2[25157] = {X 193.0441, Y 34.5207, Z -3.8333, A 0.000, B 0.000, C 0.000 }
gfCNCPoint2[25158] = {X 193.3799, Y 33.8524, Z -3.8333, A 0.000, B 0.000, C 0.000 }
gfCNCPoint2[25159] = {X 193.4229, Y 33.7850, Z -3.8333, A 0.000, B 0.000, C 0.000 }
gfCNCPoint2[25160] = {X 193.4672, Y 33.7184, Z -3.8333, A 0.000, B 0.000, C 0.000 }
gfCNCPoint2[25161] = {X 193.3656, Y 33.7152, Z -3.8333, A 0.000, B 0.000, C 0.000 }
gfCNCPoint2[25162] = {X 192.6816, Y 33.8774, Z -3.8333, A 0.000, B 0.000, C 0.000 }
gfCNCPoint2[25163] = {X 190.9512, Y 34.1514, Z -3.8333, A 0.000, B 0.000, C 0.000 }
gfCNCPoint2[25164] = {X 189.2078, Y 34.3245, Z -3.8333, A 0.000, B 0.000, C 0.000 }
gfCNCPoint2[25165] = {X 186.9429, Y 34.4635, Z -3.8333, A 0.000, B 0.000, C 0.000 }
gfCNCPoint2[25166] = {X 182.9870, Y 35.0557, Z -3.8333, A 0.000, B 0.000, C 0.000 }
gfCNCPoint2[25167] = {X 190.9367, Y 34.4874, Z -3.8333, A 0.000, B 0.000, C 0.000 }
gfCNCPoint2[25168] = {X 186.9380, Y 34.3837, Z -3.8333, A 0.000, B 0.000, C 0.000 }
gfCNCPoint2[25169] = {X 182.5512, Y 34.6530, Z -3.8333, A 0.000, B 0.000, C 0.000 }
gfCNCPoint2[25170] = {X 181.6423, Y 34.7646, Z -3.8333, A 0.000, B 0.000, C 0.000 }
gfCNCPoint2[25171] = {X 180.7536, Y 34.9855, Z -3.8333, A 0.000, B 0.000, C 0.000 }
gfCNCPoint2[25172] = {X 180.6822, Y 35.2184, Z -3.8333, A 0.000, B 0.000, C 0.000 }
gfCNCPoint2[25173] = {X 180.6645, Y 35.4613, Z -3.8333, A 0.000, B 0.000, C 0.000 }
gfCNCPoint2[25174] = {X 180.7791, Y 36.1302, Z -3.8333, A 0.000, B 0.000, C 0.000 }
gfCNCPoint2[25175] = {X 181.0966, Y 36.7299, Z -3.8333, A 0.000, B 0.000, C 0.000 }
gfCNCPoint2[25176] = {X 181.5852, Y 37.2008, Z -3.8333, A 0.000, B 0.000, C 0.000 }
gfCNCPoint2[25177] = {X 182.2545, Y 37.5834, Z -3.8333, A 0.000, B 0.000, C 0.000 }
gfCNCPoint2[25178] = {X 182.9702, Y 37.8700, Z -3.8333, A 0.000, B 0.000, C 0.000 }
gfCNCPoint2[25179] = {X 184.4318, Y 38.1967, Z -3.8333, A 0.000, B 0.000, C 0.000 }
gfCNCPoint2[25180] = {X 185.9247, Y 38.3175, Z -3.8333, A 0.000, B 0.000, C 0.000 }
gfCNCPoint2[25181] = {X 187.4198, Y 38.2301, Z -3.8333, A 0.000, B 0.000, C 0.000 }
gfCNCPoint2[25182] = {X 188.8884, Y 37.9361, Z -3.8333, A 0.000, B 0.000, C 0.000 }
gfCNCPoint2[25183] = {X 190.3020, Y 37.4413, Z -3.8333, A 0.000, B 0.000, C 0.000 }
gfCNCPoint2[25184] = {X 191.6084, Y 36.7982, Z -3.8333, A 0.000, B 0.000, C 0.000 }
gfCNCPoint2[25185] = {X 192.8422, Y 36.0250, Z -3.8333, A 0.000, B 0.000, C 0.000 }
gfCNCPoint2[25186] = {X 192.9290, Y 35.1818, Z -3.8333, A 0.000, B 0.000, C 0.000 }
gfCNCPoint2[25187] = {X 193.1917, Y 34.3757, Z -3.8333, A 0.000, B 0.000, C 0.000 }
gfCNCPoint2[25188] = {X 193.6183, Y 33.6431, Z -3.8333, A 0.000, B 0.000, C 0.000 }
gfCNCPoint2[25189] = {X 193.3575, Y 33.6349, Z -3.8333, A 0.000, B 0.000, C 0.000 }
gfCNCPoint2[25190] = {X 192.6650, Y 33.7991, Z -3.8333, A 0.000, B 0.000, C 0.000 }
